LIN {X 0,Y 574.636,Z 652.296,A -85,B 0,C 180,E1 -2267.181,E2 -2267.181} C_VEL
LIN {X 0,Y 574.744,Z 636.733,A -85,B 0,C 180,E1 -2267.487,E2 -2267.487} C_VEL
LIN {X 0,Y 575.18,Z 481.073,A -85,B 0,C 180,E1 -2269.488,E2 -2269.488} C_VEL
LIN {X 0,Y 574.004,Z 474.783,A -85,B 0,C 180,E1 -2269.626,E2 -2269.626} C_VEL
LIN {X 0,Y 574.349,Z 449.397,A -85,B 0,C 180,E1 -2272.671,E2 -2272.671} C_VEL
LIN {X 0,Y 574.64,Z 427.548,A -85,B 0,C 180,E1 -2275.344,E2 -2275.344} C_VEL
LIN {X 0,Y 574.378,Z 424.427,A -85,B 0,C 180,E1 -2275.745,E2 -2275.745} C_VEL
LIN {X 0,Y 573.261,Z 419.708,A -85,B 0,C 180,E1 -2276.421,E2 -2276.421} C_VEL
LIN {X 0,Y 573.237,Z 419.708,A -85,B 0,C 180,E1 -2278.564,E2 -2278.564} C_VEL
LIN {X 0,Y 573.234,Z 419.702,A -85,B 0,C 180,E1 -2280.992,E2 -2280.992} C_VEL
LIN {X 0,Y 573.259,Z 419.698,A -85,B 0,C 180,E1 -2283.523,E2 -2283.523} C_VEL
LIN {X 0,Y 573.241,Z 419.705,A -85,B 0,C 180,E1 -2286.049,E2 -2286.049} C_VEL
LIN {X 0,Y 573.245,Z 419.702,A -85,B 0,C 180,E1 -2288.7,E2 -2288.7} C_VEL
LIN {X 0,Y 573.249,Z 419.699,A -85,B 0,C 180,E1 -2291.595,E2 -2291.595} C_VEL
LIN {X 0,Y 573.234,Z 419.71,A -85,B 0,C 180,E1 -2294.332,E2 -2294.332} C_VEL
LIN {X 0,Y 573.234,Z 419.699,A -85,B 0,C 180,E1 -2297.358,E2 -2297.358} C_VEL
LIN {X 0,Y 573.243,Z 419.708,A -85,B 0,C 180,E1 -2300.393,E2 -2300.393} C_VEL
LIN {X 0,Y 573.25,Z 419.698,A -85,B 0,C 180,E1 -2303.077,E2 -2303.077} C_VEL
LIN {X 0,Y 573.268,Z 419.697,A -85,B 0,C 180,E1 -2305.672,E2 -2305.672} C_VEL
LIN {X 0,Y 573.243,Z 419.706,A -85,B 0,C 180,E1 -2308.185,E2 -2308.185} C_VEL
LIN {X 0,Y 573.26,Z 419.702,A -85,B 0,C 180,E1 -2310.634,E2 -2310.634} C_VEL
LIN {X 0,Y 573.264,Z 419.696,A -85,B 0,C 180,E1 -2313.5,E2 -2313.5} C_VEL
LIN {X 0,Y 573.226,Z 419.707,A -85,B 0,C 180,E1 -2316.134,E2 -2316.134} C_VEL
LIN {X 0,Y 573.254,Z 419.697,A -85,B 0,C 180,E1 -2319.174,E2 -2319.174} C_VEL
LIN {X 0,Y 573.231,Z 419.7,A -85,B 0,C 180,E1 -2321.412,E2 -2321.412} C_VEL
LIN {X 0,Y 573.252,Z 419.697,A -85,B 0,C 180,E1 -2323.622,E2 -2323.622} C_VEL
LIN {X 0,Y 573.23,Z 419.707,A -85,B 0,C 180,E1 -2326.53,E2 -2326.53} C_VEL
LIN {X 0,Y 573.254,Z 419.701,A -85,B 0,C 180,E1 -2328.745,E2 -2328.745} C_VEL
LIN {X 0,Y 573.301,Z 419.691,A -85,B 0,C 180,E1 -2331.541,E2 -2331.541} C_VEL
LIN {X 0,Y 573.284,Z 419.703,A -85,B 0,C 180,E1 -2334.372,E2 -2334.372} C_VEL
LIN {X 0,Y 573.304,Z 419.693,A -85,B 0,C 180,E1 -2337.893,E2 -2337.893} C_VEL
LIN {X 0,Y 573.329,Z 419.692,A -85,B 0,C 180,E1 -2340.703,E2 -2340.703} C_VEL
LIN {X 0,Y 573.234,Z 419.7,A -85,B 0,C 180,E1 -2343.515,E2 -2343.515} C_VEL
LIN {X 0,Y 573.291,Z 419.693,A -85,B 0,C 180,E1 -2345.628,E2 -2345.628} C_VEL
LIN {X 0,Y 573.301,Z 419.701,A -85,B 0,C 180,E1 -2348.459,E2 -2348.459} C_VEL
LIN {X 0,Y 573.264,Z 419.695,A -85,B 0,C 180,E1 -2351.312,E2 -2351.312} C_VEL
LIN {X 0,Y 573.266,Z 419.702,A -85,B 0,C 180,E1 -2354.193,E2 -2354.193} C_VEL
LIN {X 0,Y 573.254,Z 419.698,A -85,B 0,C 180,E1 -2357.112,E2 -2357.112} C_VEL
LIN {X 0,Y 573.252,Z 419.702,A -85,B 0,C 180,E1 -2360.077,E2 -2360.077} C_VEL
LIN {X 0,Y 573.236,Z 419.709,A -85,B 0,C 180,E1 -2362.338,E2 -2362.338} C_VEL
LIN {X 0,Y 573.246,Z 419.703,A -85,B 0,C 180,E1 -2364.399,E2 -2364.399} C_VEL
LIN {X 0,Y 572.62,Z 419.784,A -85,B 0,C 180,E1 -2364.986,E2 -2364.986} C_VEL
LIN {X 0,Y 569.782,Z 420.136,A -85,B 0,C 180,E1 -2365.938,E2 -2365.938} C_VEL
LIN {X 0,Y 567.354,Z 420.438,A -85,B 0,C 180,E1 -2366.704,E2 -2366.704} C_VEL
LIN {X 0,Y 566.301,Z 420.564,A -85,B 0,C 180,E1 -2367.295,E2 -2367.295} C_VEL
LIN {X 0,Y 566.212,Z 420.575,A -85,B 0,C 180,E1 -2367.495,E2 -2367.495} C_VEL
LIN {X 0,Y 566.223,Z 420.574,A -85,B 0,C 180,E1 -2369.768,E2 -2369.768} C_VEL
LIN {X 0,Y 566.205,Z 420.584,A -85,B 0,C 180,E1 -2372.432,E2 -2372.432} C_VEL
LIN {X 0,Y 566.21,Z 420.578,A -85,B 0,C 180,E1 -2374.995,E2 -2374.995} C_VEL
LIN {X 0,Y 566.193,Z 420.578,A -85,B 0,C 180,E1 -2377.461,E2 -2377.461} C_VEL
LIN {X 0,Y 566.224,Z 420.581,A -85,B 0,C 180,E1 -2380.198,E2 -2380.198} C_VEL
LIN {X 0,Y 566.198,Z 420.582,A -85,B 0,C 180,E1 -2383.055,E2 -2383.055} C_VEL
LIN {X 0,Y 566.226,Z 420.717,A -85,B 0,C 180,E1 -2384.592,E2 -2384.592} C_VEL
LIN {X 0,Y 567.225,Z 426.295,A -85,B 0,C 180,E1 -2385.433,E2 -2385.433} C_VEL
LIN {X 0,Y 566.895,Z 445.97,A -85,B 0,C 180,E1 -2388.193,E2 -2388.193} C_VEL
LIN {X 0,Y 568.518,Z 454.109,A -85,B 0,C 180,E1 -2388.359,E2 -2388.359} C_VEL
LIN {X 0,Y 567.983,Z 611.267,A -85,B 0,C 180,E1 -2390.415,E2 -2390.415} C_VEL
LIN {X 0,Y 567.818,Z 627.039,A -85,B 0,C 180,E1 -2390.774,E2 -2390.774} C_VEL
LIN {X 0,Y 567.61,Z 641.985,A -85,B 0,C 180,E1 -2391.265,E2 -2391.265} C_VEL
LIN {X 0,Y 567.394,Z 656.381,A -85,B 0,C 180,E1 -2391.892,E2 -2391.892} C_VEL
LIN {X 0,Y 567.139,Z 669.582,A -85,B 0,C 180,E1 -2392.613,E2 -2392.613} C_VEL
LIN {X 0,Y 566.915,Z 682.658,A -85,B 0,C 180,E1 -2393.485,E2 -2393.485} C_VEL
LIN {X 0,Y 566.723,Z 693.514,A -85,B 0,C 180,E1 -2394.35,E2 -2394.35} C_VEL
LIN {X 0,Y 566.452,Z 704.885,A -85,B 0,C 180,E1 -2395.416,E2 -2395.416} C_VEL
LIN {X 0,Y 566.33,Z 714.474,A -85,B 0,C 180,E1 -2396.481,E2 -2396.481} C_VEL
LIN {X 0,Y 566.203,Z 724.073,A -85,B 0,C 180,E1 -2397.743,E2 -2397.743} C_VEL
LIN {X 0,Y 566.055,Z 731.777,A -85,B 0,C 180,E1 -2398.947,E2 -2398.947} C_VEL
LIN {X 0,Y 566.009,Z 739.23,A -85,B 0,C 180,E1 -2400.363,E2 -2400.363} C_VEL
LIN {X 0,Y 565.929,Z 745.455,A -85,B 0,C 180,E1 -2401.85,E2 -2401.85} C_VEL
LIN {X 0,Y 565.901,Z 750.37,A -85,B 0,C 180,E1 -2403.404,E2 -2403.404} C_VEL
LIN {X 0,Y 565.853,Z 753.908,A -85,B 0,C 180,E1 -2405.022,E2 -2405.022} C_VEL
LIN {X 0,Y 565.848,Z 755.883,A -85,B 0,C 180,E1 -2406.582,E2 -2406.582} C_VEL
LIN {X 0,Y 565.831,Z 756.489,A -85,B 0,C 180,E1 -2408.123,E2 -2408.123} C_VEL
LIN {X 0,Y 565.833,Z 755.776,A -85,B 0,C 180,E1 -2409.649,E2 -2409.649} C_VEL
LIN {X 0,Y 565.851,Z 753.765,A -85,B 0,C 180,E1 -2411.161,E2 -2411.161} C_VEL
LIN {X 0,Y 565.862,Z 750.442,A -85,B 0,C 180,E1 -2412.658,E2 -2412.658} C_VEL
LIN {X 0,Y 565.916,Z 745.782,A -85,B 0,C 180,E1 -2414.145,E2 -2414.145} C_VEL
LIN {X 0,Y 566.005,Z 739.706,A -85,B 0,C 180,E1 -2415.621,E2 -2415.621} C_VEL
LIN {X 0,Y 566.037,Z 732.099,A -85,B 0,C 180,E1 -2417.086,E2 -2417.086} C_VEL
LIN {X 0,Y 566.205,Z 723.96,A -85,B 0,C 180,E1 -2418.364,E2 -2418.364} C_VEL
LIN {X 0,Y 566.34,Z 714.266,A -85,B 0,C 180,E1 -2419.634,E2 -2419.634} C_VEL
LIN {X 0,Y 566.521,Z 704.419,A -85,B 0,C 180,E1 -2420.72,E2 -2420.72} C_VEL
LIN {X 0,Y 566.736,Z 692.793,A -85,B 0,C 180,E1 -2421.802,E2 -2421.802} C_VEL
LIN {X 0,Y 566.935,Z 680.459,A -85,B 0,C 180,E1 -2422.762,E2 -2422.762} C_VEL
LIN {X 0,Y 567.195,Z 667.503,A -85,B 0,C 180,E1 -2423.598,E2 -2423.598} C_VEL
LIN {X 0,Y 567.46,Z 653.878,A -85,B 0,C 180,E1 -2424.314,E2 -2424.314} C_VEL
LIN {X 0,Y 567.64,Z 640.029,A -85,B 0,C 180,E1 -2424.895,E2 -2424.895} C_VEL
LIN {X 0,Y 567.851,Z 625.202,A -85,B 0,C 180,E1 -2425.364,E2 -2425.364} C_VEL
LIN {X 0,Y 567.962,Z 609.905,A -85,B 0,C 180,E1 -2425.698,E2 -2425.698} C_VEL
LIN {X 0,Y 568.45,Z 453.464,A -85,B 0,C 180,E1 -2427.742,E2 -2427.742} C_VEL
LIN {X 0,Y 566.942,Z 445.815,A -85,B 0,C 180,E1 -2427.914,E2 -2427.914} C_VEL
LIN {X 0,Y 567.186,Z 425.932,A -85,B 0,C 180,E1 -2430.71,E2 -2430.71} C_VEL
LIN {X 0,Y 566.227,Z 420.583,A -85,B 0,C 180,E1 -2431.534,E2 -2431.534} C_VEL
LIN {X 0,Y 566.195,Z 420.587,A -85,B 0,C 180,E1 -2433.559,E2 -2433.559} C_VEL
LIN {X 0,Y 566.26,Z 420.577,A -85,B 0,C 180,E1 -2435.699,E2 -2435.699} C_VEL
LIN {X 0,Y 566.232,Z 420.573,A -85,B 0,C 180,E1 -2438.566,E2 -2438.566} C_VEL
LIN {X 0,Y 566.247,Z 420.575,A -85,B 0,C 180,E1 -2441.454,E2 -2441.454} C_VEL
LIN {X 0,Y 566.24,Z 420.572,A -85,B 0,C 180,E1 -2444.507,E2 -2444.507} C_VEL
LIN {X 0,Y 566.204,Z 420.581,A -85,B 0,C 180,E1 -2447.332,E2 -2447.332} C_VEL
LIN {X 0,Y 566.217,Z 420.575,A -85,B 0,C 180,E1 -2450.337,E2 -2450.337} C_VEL
LIN {X 0,Y 566.194,Z 420.583,A -85,B 0,C 180,E1 -2453.404,E2 -2453.404} C_VEL
LIN {X 0,Y 566.219,Z 420.582,A -85,B 0,C 180,E1 -2455.749,E2 -2455.749} C_VEL
LIN {X 0,Y 566.207,Z 420.576,A -85,B 0,C 180,E1 -2458.202,E2 -2458.202} C_VEL
LIN {X 0,Y 566.203,Z 420.578,A -85,B 0,C 180,E1 -2461.078,E2 -2461.078} C_VEL
LIN {X 0,Y 566.215,Z 420.583,A -85,B 0,C 180,E1 -2463.734,E2 -2463.734} C_VEL
LIN {X 0,Y 566.218,Z 420.573,A -85,B 0,C 180,E1 -2466.569,E2 -2466.569} C_VEL
LIN {X 0,Y 566.215,Z 420.584,A -85,B 0,C 180,E1 -2469.685,E2 -2469.685} C_VEL
LIN {X 0,Y 566.217,Z 420.576,A -85,B 0,C 180,E1 -2472.087,E2 -2472.087} C_VEL
LIN {X 0,Y 566.176,Z 420.58,A -85,B 0,C 180,E1 -2475.036,E2 -2475.036} C_VEL
LIN {X 0,Y 566.214,Z 420.575,A -85,B 0,C 180,E1 -2478.136,E2 -2478.136} C_VEL
LIN {X 0,Y 566.224,Z 420.573,A -85,B 0,C 180,E1 -2480.727,E2 -2480.727} C_VEL
LIN {X 0,Y 566.22,Z 420.58,A -85,B 0,C 180,E1 -2483.783,E2 -2483.783} C_VEL
LIN {X 0,Y 566.214,Z 420.576,A -85,B 0,C 180,E1 -2486.265,E2 -2486.265} C_VEL
LIN {X 0,Y 566.192,Z 420.577,A -85,B 0,C 180,E1 -2488.923,E2 -2488.923} C_VEL
LIN {X 0,Y 566.23,Z 420.579,A -85,B 0,C 180,E1 -2491.858,E2 -2491.858} C_VEL
LIN {X 0,Y 566.226,Z 420.574,A -85,B 0,C 180,E1 -2494.251,E2 -2494.251} C_VEL
LIN {X 0,Y 566.173,Z 420.576,A -85,B 0,C 180,E1 -2496.718,E2 -2496.718} C_VEL
LIN {X 0,Y 566.215,Z 420.584,A -85,B 0,C 180,E1 -2499.663,E2 -2499.663} C_VEL
LIN {X 0,Y 566.2,Z 420.574,A -85,B 0,C 180,E1 -2502.668,E2 -2502.668} C_VEL
LIN {X 0,Y 566.234,Z 420.58,A -85,B 0,C 180,E1 -2505.627,E2 -2505.627} C_VEL
LIN {X 0,Y 566.234,Z 420.57,A -85,B 0,C 180,E1 -2508.675,E2 -2508.675} C_VEL
LIN {X 0,Y 566.234,Z 420.575,A -85,B 0,C 180,E1 -2511.434,E2 -2511.434} C_VEL
LIN {X 0,Y 566.258,Z 420.57,A -85,B 0,C 180,E1 -2514.301,E2 -2514.301} C_VEL
LIN {X 0,Y 566.28,Z 420.572,A -85,B 0,C 180,E1 -2517.866,E2 -2517.866} C_VEL
LIN {X 0,Y 566.303,Z 420.563,A -85,B 0,C 180,E1 -2520.711,E2 -2520.711} C_VEL
LIN {X 0,Y 566.275,Z 420.566,A -85,B 0,C 180,E1 -2522.845,E2 -2522.845} C_VEL
LIN {X 0,Y 566.257,Z 420.576,A -85,B 0,C 180,E1 -2525.698,E2 -2525.698} C_VEL
LIN {X 0,Y 566.233,Z 420.572,A -85,B 0,C 180,E1 -2528.565,E2 -2528.565} C_VEL
LIN {X 0,Y 566.241,Z 420.575,A -85,B 0,C 180,E1 -2531.454,E2 -2531.454} C_VEL
LIN {X 0,Y 566.233,Z 420.572,A -85,B 0,C 180,E1 -2534.506,E2 -2534.506} C_VEL
LIN {X 0,Y 566.199,Z 420.58,A -85,B 0,C 180,E1 -2537.331,E2 -2537.331} C_VEL
LIN {X 0,Y 566.213,Z 420.576,A -85,B 0,C 180,E1 -2540.337,E2 -2540.337} C_VEL
LIN {X 0,Y 566.188,Z 420.582,A -85,B 0,C 180,E1 -2543.404,E2 -2543.404} C_VEL
LIN {X 0,Y 566.215,Z 420.584,A -85,B 0,C 180,E1 -2545.749,E2 -2545.749} C_VEL
LIN {X 0,Y 566.205,Z 420.578,A -85,B 0,C 180,E1 -2548.203,E2 -2548.203} C_VEL
LIN {X 0,Y 566.189,Z 420.578,A -85,B 0,C 180,E1 -2551.076,E2 -2551.076} C_VEL
LIN {X 0,Y 566.212,Z 420.584,A -85,B 0,C 180,E1 -2553.734,E2 -2553.734} C_VEL
LIN {X 0,Y 566.216,Z 420.574,A -85,B 0,C 180,E1 -2556.569,E2 -2556.569} C_VEL
LIN {X 0,Y 566.211,Z 420.585,A -85,B 0,C 180,E1 -2559.685,E2 -2559.685} C_VEL
LIN {X 0,Y 566.188,Z 420.582,A -85,B 0,C 180,E1 -2562.09,E2 -2562.09} C_VEL
LIN {X 0,Y 566.174,Z 420.58,A -85,B 0,C 180,E1 -2565.036,E2 -2565.036} C_VEL
LIN {X 0,Y 566.214,Z 420.582,A -85,B 0,C 180,E1 -2567.913,E2 -2567.913} C_VEL
LIN {X 0,Y 566.217,Z 420.574,A -85,B 0,C 180,E1 -2570.727,E2 -2570.727} C_VEL
LIN {X 0,Y 566.184,Z 420.587,A -85,B 0,C 180,E1 -2573.788,E2 -2573.788} C_VEL
LIN {X 0,Y 566.212,Z 420.579,A -85,B 0,C 180,E1 -2576.266,E2 -2576.266} C_VEL
LIN {X 0,Y 566.196,Z 420.579,A -85,B 0,C 180,E1 -2578.923,E2 -2578.923} C_VEL
LIN {X 0,Y 566.212,Z 420.585,A -85,B 0,C 180,E1 -2581.857,E2 -2581.857} C_VEL
LIN {X 0,Y 566.204,Z 420.669,A -85,B 0,C 180,E1 -2583.394,E2 -2583.394} C_VEL
LIN {X 0,Y 567.792,Z 427.532,A -85,B 0,C 180,E1 -2584.328,E2 -2584.328} C_VEL
LIN {X 0,Y 567.557,Z 447.83,A -85,B 0,C 180,E1 -2586.849,E2 -2586.849} C_VEL
LIN {X 0,Y 567.148,Z 472.644,A -85,B 0,C 180,E1 -2589.868,E2 -2589.868} C_VEL
LIN {X 0,Y 567.114,Z 474.917,A -85,B 0,C 180,E1 -2590.142,E2 -2590.142} C_VEL
LIN {X 0,Y 568.492,Z 482.253,A -85,B 0,C 180,E1 -2590.289,E2 -2590.289} C_VEL
LIN {X 0,Y 567.986,Z 640.908,A -85,B 0,C 180,E1 -2592.363,E2 -2592.363} C_VEL
LIN {X 0,Y 567.836,Z 656.698,A -85,B 0,C 180,E1 -2592.72,E2 -2592.72} C_VEL
LIN {X 0,Y 567.632,Z 672.035,A -85,B 0,C 180,E1 -2593.223,E2 -2593.223} C_VEL
LIN {X 0,Y 567.459,Z 685.767,A -85,B 0,C 180,E1 -2593.819,E2 -2593.819} C_VEL
LIN {X 0,Y 567.151,Z 699.241,A -85,B 0,C 180,E1 -2594.548,E2 -2594.548} C_VEL
LIN {X 0,Y 566.932,Z 711.516,A -85,B 0,C 180,E1 -2595.359,E2 -2595.359} C_VEL
LIN {X 0,Y 566.672,Z 724.287,A -85,B 0,C 180,E1 -2596.37,E2 -2596.37} C_VEL
LIN {X 0,Y 566.491,Z 735.746,A -85,B 0,C 180,E1 -2597.461,E2 -2597.461} C_VEL
LIN {X 0,Y 566.269,Z 746.31,A -85,B 0,C 180,E1 -2598.659,E2 -2598.659} C_VEL
LIN {X 0,Y 566.208,Z 754.855,A -85,B 0,C 180,E1 -2599.812,E2 -2599.812} C_VEL
LIN {X 0,Y 566.058,Z 762.732,A -85,B 0,C 180,E1 -2601.072,E2 -2601.072} C_VEL
LIN {X 0,Y 565.998,Z 770.088,A -85,B 0,C 180,E1 -2602.508,E2 -2602.508} C_VEL
LIN {X 0,Y 565.956,Z 775.922,A -85,B 0,C 180,E1 -2603.941,E2 -2603.941} C_VEL
LIN {X 0,Y 565.866,Z 779.384,A -85,B 0,C 180,E1 -2605.012,E2 -2605.012} C_VEL
LIN {X 0,Y 565.909,Z 782.889,A -85,B 0,C 180,E1 -2606.44,E2 -2606.44} C_VEL
LIN {X 0,Y 565.836,Z 785.192,A -85,B 0,C 180,E1 -2607.864,E2 -2607.864} C_VEL
LIN {X 0,Y 565.838,Z 786.349,A -85,B 0,C 180,E1 -2609.288,E2 -2609.288} C_VEL
LIN {X 0,Y 565.838,Z 786.349,A -85,B 0,C 180,E1 -2610.711,E2 -2610.711} C_VEL
LIN {X 0,Y 565.836,Z 785.191,A -85,B 0,C 180,E1 -2612.135,E2 -2612.135} C_VEL
LIN {X 0,Y 565.909,Z 782.888,A -85,B 0,C 180,E1 -2613.56,E2 -2613.56} C_VEL
LIN {X 0,Y 565.866,Z 779.387,A -85,B 0,C 180,E1 -2614.987,E2 -2614.987} C_VEL
LIN {X 0,Y 565.956,Z 775.926,A -85,B 0,C 180,E1 -2616.059,E2 -2616.059} C_VEL
LIN {X 0,Y 565.999,Z 770.09,A -85,B 0,C 180,E1 -2617.491,E2 -2617.491} C_VEL
LIN {X 0,Y 566.057,Z 762.733,A -85,B 0,C 180,E1 -2618.928,E2 -2618.928} C_VEL
LIN {X 0,Y 566.208,Z 754.86,A -85,B 0,C 180,E1 -2620.187,E2 -2620.187} C_VEL
LIN {X 0,Y 566.307,Z 745.395,A -85,B 0,C 180,E1 -2621.452,E2 -2621.452} C_VEL
LIN {X 0,Y 566.491,Z 735.754,A -85,B 0,C 180,E1 -2622.539,E2 -2622.539} C_VEL
LIN {X 0,Y 566.671,Z 724.3,A -85,B 0,C 180,E1 -2623.629,E2 -2623.629} C_VEL
LIN {X 0,Y 566.926,Z 711.683,A -85,B 0,C 180,E1 -2624.63,E2 -2624.63} C_VEL
LIN {X 0,Y 567.123,Z 699.253,A -85,B 0,C 180,E1 -2625.452,E2 -2625.452} C_VEL
LIN {X 0,Y 567.418,Z 685.779,A -85,B 0,C 180,E1 -2626.181,E2 -2626.181} C_VEL
LIN {X 0,Y 567.606,Z 672.062,A -85,B 0,C 180,E1 -2626.777,E2 -2626.777} C_VEL
LIN {X 0,Y 567.845,Z 656.738,A -85,B 0,C 180,E1 -2627.279,E2 -2627.279} C_VEL
LIN {X 0,Y 567.978,Z 641.331,A -85,B 0,C 180,E1 -2627.629,E2 -2627.629} C_VEL
LIN {X 0,Y 568.463,Z 481.789,A -85,B 0,C 180,E1 -2629.718,E2 -2629.718} C_VEL
LIN {X 0,Y 567.132,Z 474.839,A -85,B 0,C 180,E1 -2629.867,E2 -2629.867} C_VEL
LIN {X 0,Y 567.488,Z 449.397,A -85,B 0,C 180,E1 -2632.961,E2 -2632.961} C_VEL
LIN {X 0,Y 567.849,Z 429.252,A -85,B 0,C 180,E1 -2635.454,E2 -2635.454} C_VEL
LIN {X 0,Y 567.492,Z 425.948,A -85,B 0,C 180,E1 -2635.883,E2 -2635.883} C_VEL
LIN {X 0,Y 566.205,Z 420.587,A -85,B 0,C 180,E1 -2636.626,E2 -2636.626} C_VEL
LIN {X 0,Y 566.19,Z 420.582,A -85,B 0,C 180,E1 -2638.953,E2 -2638.953} C_VEL
LIN {X 0,Y 566.199,Z 420.578,A -85,B 0,C 180,E1 -2641.421,E2 -2641.421} C_VEL
LIN {X 0,Y 566.206,Z 420.581,A -85,B 0,C 180,E1 -2643.955,E2 -2643.955} C_VEL
LIN {X 0,Y 566.208,Z 420.581,A -85,B 0,C 180,E1 -2646.568,E2 -2646.568} C_VEL
LIN {X 0,Y 566.209,Z 420.577,A -85,B 0,C 180,E1 -2649.685,E2 -2649.685} C_VEL
LIN {X 0,Y 566.212,Z 420.582,A -85,B 0,C 180,E1 -2652.086,E2 -2652.086} C_VEL
LIN {X 0,Y 566.168,Z 420.581,A -85,B 0,C 180,E1 -2655.035,E2 -2655.035} C_VEL
LIN {X 0,Y 566.212,Z 420.581,A -85,B 0,C 180,E1 -2658.135,E2 -2658.135} C_VEL
LIN {X 0,Y 566.217,Z 420.578,A -85,B 0,C 180,E1 -2660.727,E2 -2660.727} C_VEL
LIN {X 0,Y 566.212,Z 420.577,A -85,B 0,C 180,E1 -2663.783,E2 -2663.783} C_VEL
LIN {X 0,Y 566.223,Z 420.583,A -85,B 0,C 180,E1 -2666.263,E2 -2666.263} C_VEL
LIN {X 0,Y 566.192,Z 420.578,A -85,B 0,C 180,E1 -2668.922,E2 -2668.922} C_VEL
LIN {X 0,Y 566.221,Z 420.576,A -85,B 0,C 180,E1 -2671.858,E2 -2671.858} C_VEL
LIN {X 0,Y 566.22,Z 420.582,A -85,B 0,C 180,E1 -2674.251,E2 -2674.251} C_VEL
LIN {X 0,Y 566.184,Z 420.582,A -85,B 0,C 180,E1 -2676.713,E2 -2676.713} C_VEL
LIN {X 0,Y 566.212,Z 420.575,A -85,B 0,C 180,E1 -2679.663,E2 -2679.663} C_VEL
LIN {X 0,Y 566.197,Z 420.58,A -85,B 0,C 180,E1 -2682.668,E2 -2682.668} C_VEL
LIN {X 0,Y 566.226,Z 420.573,A -85,B 0,C 180,E1 -2685.627,E2 -2685.627} C_VEL
LIN {X 0,Y 566.226,Z 420.577,A -85,B 0,C 180,E1 -2688.675,E2 -2688.675} C_VEL
LIN {X 0,Y 566.242,Z 420.57,A -85,B 0,C 180,E1 -2691.435,E2 -2691.435} C_VEL
LIN {X 0,Y 566.252,Z 420.578,A -85,B 0,C 180,E1 -2694.302,E2 -2694.302} C_VEL
LIN {X 0,Y 566.275,Z 420.568,A -85,B 0,C 180,E1 -2697.866,E2 -2697.866} C_VEL
LIN {X 0,Y 566.299,Z 420.567,A -85,B 0,C 180,E1 -2700.711,E2 -2700.711} C_VEL
LIN {X 0,Y 566.272,Z 420.57,A -85,B 0,C 180,E1 -2702.846,E2 -2702.846} C_VEL
LIN {X 0,Y 566.26,Z 420.569,A -85,B 0,C 180,E1 -2705.698,E2 -2705.698} C_VEL
LIN {X 0,Y 566.242,Z 420.578,A -85,B 0,C 180,E1 -2708.566,E2 -2708.566} C_VEL
LIN {X 0,Y 566.234,Z 420.571,A -85,B 0,C 180,E1 -2711.455,E2 -2711.455} C_VEL
LIN {X 0,Y 566.227,Z 420.581,A -85,B 0,C 180,E1 -2714.507,E2 -2714.507} C_VEL
LIN {X 0,Y 566.199,Z 420.576,A -85,B 0,C 180,E1 -2717.332,E2 -2717.332} C_VEL
LIN {X 0,Y 566.214,Z 420.583,A -85,B 0,C 180,E1 -2720.337,E2 -2720.337} C_VEL
LIN {X 0,Y 566.185,Z 420.578,A -85,B 0,C 180,E1 -2723.404,E2 -2723.404} C_VEL
LIN {X 0,Y 566.222,Z 420.575,A -85,B 0,C 180,E1 -2725.749,E2 -2725.749} C_VEL
LIN {X 0,Y 566.212,Z 420.575,A -85,B 0,C 180,E1 -2727.495,E2 -2727.495} C_VEL
LIN {X 0,Y 565.534,Z 420.666,A -85,B 0,C 180,E1 -2728.089,E2 -2728.089} C_VEL
LIN {X 0,Y 562.669,Z 421.02,A -85,B 0,C 180,E1 -2729.053,E2 -2729.053} C_VEL
LIN {X 0,Y 560.258,Z 421.32,A -85,B 0,C 180,E1 -2729.828,E2 -2729.828} C_VEL
LIN {X 0,Y 559.229,Z 421.453,A -85,B 0,C 180,E1 -2730.427,E2 -2730.427} C_VEL
LIN {X 0,Y 559.148,Z 421.457,A -85,B 0,C 180,E1 -2730.63,E2 -2730.63} C_VEL
LIN {X 0,Y 559.174,Z 421.452,A -85,B 0,C 180,E1 -2733.574,E2 -2733.574} C_VEL
LIN {X 0,Y 559.186,Z 421.459,A -85,B 0,C 180,E1 -2736.452,E2 -2736.452} C_VEL
LIN {X 0,Y 559.175,Z 421.456,A -85,B 0,C 180,E1 -2738.934,E2 -2738.934} C_VEL
LIN {X 0,Y 559.188,Z 421.452,A -85,B 0,C 180,E1 -2741.768,E2 -2741.768} C_VEL
LIN {X 0,Y 559.173,Z 421.48,A -85,B 0,C 180,E1 -2744.381,E2 -2744.381} C_VEL
LIN {X 0,Y 560.333,Z 427.983,A -85,B 0,C 180,E1 -2745.383,E2 -2745.383} C_VEL
LIN {X 0,Y 560.011,Z 446.073,A -85,B 0,C 180,E1 -2747.94,E2 -2747.94} C_VEL
LIN {X 0,Y 561.851,Z 454.621,A -85,B 0,C 180,E1 -2748.122,E2 -2748.122} C_VEL
LIN {X 0,Y 561.246,Z 610.539,A -85,B 0,C 180,E1 -2750.183,E2 -2750.183} C_VEL
LIN {X 0,Y 561.067,Z 625.756,A -85,B 0,C 180,E1 -2750.524,E2 -2750.524} C_VEL
LIN {X 0,Y 560.791,Z 641.157,A -85,B 0,C 180,E1 -2751.024,E2 -2751.024} C_VEL
LIN {X 0,Y 560.602,Z 655.412,A -85,B 0,C 180,E1 -2751.644,E2 -2751.644} C_VEL
LIN {X 0,Y 560.268,Z 669.518,A -85,B 0,C 180,E1 -2752.415,E2 -2752.415} C_VEL
LIN {X 0,Y 560.003,Z 681.869,A -85,B 0,C 180,E1 -2753.243,E2 -2753.243} C_VEL
LIN {X 0,Y 559.772,Z 693.455,A -85,B 0,C 180,E1 -2754.171,E2 -2754.171} C_VEL
LIN {X 0,Y 559.498,Z 704.848,A -85,B 0,C 180,E1 -2755.253,E2 -2755.253} C_VEL
LIN {X 0,Y 559.29,Z 715.295,A -85,B 0,C 180,E1 -2756.435,E2 -2756.435} C_VEL
LIN {X 0,Y 559.137,Z 724.751,A -85,B 0,C 180,E1 -2757.711,E2 -2757.711} C_VEL
LIN {X 0,Y 558.996,Z 732.557,A -85,B 0,C 180,E1 -2758.972,E2 -2758.972} C_VEL
LIN {X 0,Y 558.921,Z 739.865,A -85,B 0,C 180,E1 -2760.408,E2 -2760.408} C_VEL
LIN {X 0,Y 558.852,Z 745.129,A -85,B 0,C 180,E1 -2761.68,E2 -2761.68} C_VEL
LIN {X 0,Y 558.819,Z 750.115,A -85,B 0,C 180,E1 -2763.245,E2 -2763.245} C_VEL
LIN {X 0,Y 558.764,Z 753.784,A -85,B 0,C 180,E1 -2764.905,E2 -2764.905} C_VEL
LIN {X 0,Y 558.759,Z 755.949,A -85,B 0,C 180,E1 -2766.663,E2 -2766.663} C_VEL
LIN {X 0,Y 558.724,Z 756.46,A -85,B 0,C 180,E1 -2767.83,E2 -2767.83} C_VEL
LIN {X 0,Y 558.743,Z 755.982,A -85,B 0,C 180,E1 -2769.379,E2 -2769.379} C_VEL
LIN {X 0,Y 558.778,Z 754.211,A -85,B 0,C 180,E1 -2770.913,E2 -2770.913} C_VEL
LIN {X 0,Y 558.765,Z 751.149,A -85,B 0,C 180,E1 -2772.431,E2 -2772.431} C_VEL
LIN {X 0,Y 558.823,Z 746.756,A -85,B 0,C 180,E1 -2773.938,E2 -2773.938} C_VEL
LIN {X 0,Y 558.917,Z 740.963,A -85,B 0,C 180,E1 -2775.435,E2 -2775.435} C_VEL
LIN {X 0,Y 558.981,Z 733.656,A -85,B 0,C 180,E1 -2776.921,E2 -2776.921} C_VEL
LIN {X 0,Y 559.137,Z 725.854,A -85,B 0,C 180,E1 -2778.215,E2 -2778.215} C_VEL
LIN {X 0,Y 559.3,Z 716.529,A -85,B 0,C 180,E1 -2779.502,E2 -2779.502} C_VEL
LIN {X 0,Y 559.461,Z 707.123,A -85,B 0,C 180,E1 -2780.602,E2 -2780.602} C_VEL
LIN {X 0,Y 559.712,Z 695.993,A -85,B 0,C 180,E1 -2781.698,E2 -2781.698} C_VEL
LIN {X 0,Y 559.957,Z 683.762,A -85,B 0,C 180,E1 -2782.709,E2 -2782.709} C_VEL
LIN {X 0,Y 560.27,Z 670.608,A -85,B 0,C 180,E1 -2783.609,E2 -2783.609} C_VEL
LIN {X 0,Y 560.567,Z 655.887,A -85,B 0,C 180,E1 -2784.425,E2 -2784.425} C_VEL
LIN {X 0,Y 560.827,Z 641.346,A -85,B 0,C 180,E1 -2785.058,E2 -2785.058} C_VEL
LIN {X 0,Y 561.07,Z 626.158,A -85,B 0,C 180,E1 -2785.555,E2 -2785.555} C_VEL
LIN {X 0,Y 561.224,Z 611.314,A -85,B 0,C 180,E1 -2785.894,E2 -2785.894} C_VEL
LIN {X 0,Y 561.79,Z 454.392,A -85,B 0,C 180,E1 -2787.973,E2 -2787.973} C_VEL
LIN {X 0,Y 560.006,Z 445.905,A -85,B 0,C 180,E1 -2788.158,E2 -2788.158} C_VEL
LIN {X 0,Y 560.296,Z 427.911,A -85,B 0,C 180,E1 -2790.719,E2 -2790.719} C_VEL
LIN {X 0,Y 559.211,Z 421.457,A -85,B 0,C 180,E1 -2791.711,E2 -2791.711} C_VEL
LIN {X 0,Y 559.148,Z 421.464,A -85,B 0,C 180,E1 -2793.604,E2 -2793.604} C_VEL
LIN {X 0,Y 559.227,Z 421.453,A -85,B 0,C 180,E1 -2795.771,E2 -2795.771} C_VEL
LIN {X 0,Y 559.191,Z 421.451,A -85,B 0,C 180,E1 -2798.675,E2 -2798.675} C_VEL
LIN {X 0,Y 559.211,Z 421.454,A -85,B 0,C 180,E1 -2801.601,E2 -2801.601} C_VEL
LIN {X 0,Y 559.205,Z 421.448,A -85,B 0,C 180,E1 -2804.596,E2 -2804.596} C_VEL
LIN {X 0,Y 559.163,Z 421.462,A -85,B 0,C 180,E1 -2807.557,E2 -2807.557} C_VEL
LIN {X 0,Y 559.174,Z 421.458,A -85,B 0,C 180,E1 -2809.837,E2 -2809.837} C_VEL
LIN {X 0,Y 559.146,Z 421.458,A -85,B 0,C 180,E1 -2812.153,E2 -2812.153} C_VEL
LIN {X 0,Y 559.184,Z 421.452,A -85,B 0,C 180,E1 -2815.187,E2 -2815.187} C_VEL
LIN {X 0,Y 559.185,Z 421.457,A -85,B 0,C 180,E1 -2817.712,E2 -2817.712} C_VEL
LIN {X 0,Y 559.161,Z 421.455,A -85,B 0,C 180,E1 -2820.182,E2 -2820.182} C_VEL
LIN {X 0,Y 559.179,Z 421.448,A -85,B 0,C 180,E1 -2822.714,E2 -2822.714} C_VEL
LIN {X 0,Y 559.151,Z 421.459,A -85,B 0,C 180,E1 -2825.322,E2 -2825.322} C_VEL
LIN {X 0,Y 559.138,Z 421.458,A -85,B 0,C 180,E1 -2828.017,E2 -2828.017} C_VEL
LIN {X 0,Y 559.18,Z 421.451,A -85,B 0,C 180,E1 -2830.81,E2 -2830.81} C_VEL
LIN {X 0,Y 559.165,Z 421.461,A -85,B 0,C 180,E1 -2833.731,E2 -2833.731} C_VEL
LIN {X 0,Y 559.148,Z 421.454,A -85,B 0,C 180,E1 -2836.803,E2 -2836.803} C_VEL
LIN {X 0,Y 559.177,Z 421.452,A -85,B 0,C 180,E1 -2839.189,E2 -2839.189} C_VEL
LIN {X 0,Y 559.137,Z 421.46,A -85,B 0,C 180,E1 -2841.982,E2 -2841.982} C_VEL
LIN {X 0,Y 559.159,Z 421.451,A -85,B 0,C 180,E1 -2844.678,E2 -2844.678} C_VEL
LIN {X 0,Y 559.175,Z 421.456,A -85,B 0,C 180,E1 -2847.361,E2 -2847.361} C_VEL
LIN {X 0,Y 559.15,Z 421.455,A -85,B 0,C 180,E1 -2850.142,E2 -2850.142} C_VEL
LIN {X 0,Y 559.181,Z 421.452,A -85,B 0,C 180,E1 -2853.098,E2 -2853.098} C_VEL
LIN {X 0,Y 559.158,Z 421.46,A -85,B 0,C 180,E1 -2855.495,E2 -2855.495} C_VEL
LIN {X 0,Y 559.172,Z 421.451,A -85,B 0,C 180,E1 -2858.624,E2 -2858.624} C_VEL
LIN {X 0,Y 559.169,Z 421.452,A -85,B 0,C 180,E1 -2860.926,E2 -2860.926} C_VEL
LIN {X 0,Y 559.17,Z 421.456,A -85,B 0,C 180,E1 -2863.948,E2 -2863.948} C_VEL
LIN {X 0,Y 559.172,Z 421.454,A -85,B 0,C 180,E1 -2866.184,E2 -2866.184} C_VEL
LIN {X 0,Y 559.195,Z 421.449,A -85,B 0,C 180,E1 -2869.133,E2 -2869.133} C_VEL
LIN {X 0,Y 559.206,Z 421.451,A -85,B 0,C 180,E1 -2872.053,E2 -2872.053} C_VEL
LIN {X 0,Y 559.255,Z 421.441,A -85,B 0,C 180,E1 -2874.953,E2 -2874.953} C_VEL
LIN {X 0,Y 559.251,Z 421.448,A -85,B 0,C 180,E1 -2877.839,E2 -2877.839} C_VEL
LIN {X 0,Y 559.273,Z 421.439,A -85,B 0,C 180,E1 -2880.72,E2 -2880.72} C_VEL
LIN {X 0,Y 559.241,Z 421.442,A -85,B 0,C 180,E1 -2882.881,E2 -2882.881} C_VEL
LIN {X 0,Y 559.227,Z 421.452,A -85,B 0,C 180,E1 -2885.77,E2 -2885.77} C_VEL
LIN {X 0,Y 559.191,Z 421.449,A -85,B 0,C 180,E1 -2888.674,E2 -2888.674} C_VEL
LIN {X 0,Y 559.205,Z 421.454,A -85,B 0,C 180,E1 -2891.6,E2 -2891.6} C_VEL
LIN {X 0,Y 559.199,Z 421.448,A -85,B 0,C 180,E1 -2894.595,E2 -2894.595} C_VEL
LIN {X 0,Y 559.159,Z 421.46,A -85,B 0,C 180,E1 -2897.557,E2 -2897.557} C_VEL
LIN {X 0,Y 559.172,Z 421.459,A -85,B 0,C 180,E1 -2899.837,E2 -2899.837} C_VEL
LIN {X 0,Y 559.141,Z 421.458,A -85,B 0,C 180,E1 -2902.153,E2 -2902.153} C_VEL
LIN {X 0,Y 559.178,Z 421.453,A -85,B 0,C 180,E1 -2905.187,E2 -2905.187} C_VEL
LIN {X 0,Y 559.191,Z 421.459,A -85,B 0,C 180,E1 -2907.711,E2 -2907.711} C_VEL
LIN {X 0,Y 559.152,Z 421.456,A -85,B 0,C 180,E1 -2910.183,E2 -2910.183} C_VEL
LIN {X 0,Y 559.174,Z 421.451,A -85,B 0,C 180,E1 -2912.714,E2 -2912.714} C_VEL
LIN {X 0,Y 559.157,Z 421.457,A -85,B 0,C 180,E1 -2915.322,E2 -2915.322} C_VEL
LIN {X 0,Y 559.134,Z 421.461,A -85,B 0,C 180,E1 -2918.017,E2 -2918.017} C_VEL
LIN {X 0,Y 559.173,Z 421.451,A -85,B 0,C 180,E1 -2920.811,E2 -2920.811} C_VEL
LIN {X 0,Y 559.159,Z 421.463,A -85,B 0,C 180,E1 -2923.732,E2 -2923.732} C_VEL
LIN {X 0,Y 559.168,Z 421.452,A -85,B 0,C 180,E1 -2926.801,E2 -2926.801} C_VEL
LIN {X 0,Y 559.159,Z 421.456,A -85,B 0,C 180,E1 -2929.188,E2 -2929.188} C_VEL
LIN {X 0,Y 559.135,Z 421.462,A -85,B 0,C 180,E1 -2931.983,E2 -2931.983} C_VEL
LIN {X 0,Y 559.132,Z 421.458,A -85,B 0,C 180,E1 -2934.787,E2 -2934.787} C_VEL
LIN {X 0,Y 559.158,Z 421.46,A -85,B 0,C 180,E1 -2937.364,E2 -2937.364} C_VEL
LIN {X 0,Y 559.15,Z 421.462,A -85,B 0,C 180,E1 -2940.142,E2 -2940.142} C_VEL
LIN {X 0,Y 559.17,Z 421.459,A -85,B 0,C 180,E1 -2943.098,E2 -2943.098} C_VEL
LIN {X 0,Y 559.187,Z 421.563,A -85,B 0,C 180,E1 -2943.169,E2 -2943.169} C_VEL
LIN {X 0,Y 560.998,Z 429.565,A -85,B 0,C 180,E1 -2944.271,E2 -2944.271} C_VEL
LIN {X 0,Y 560.697,Z 449.39,A -85,B 0,C 180,E1 -2946.744,E2 -2946.744} C_VEL
LIN {X 0,Y 560.258,Z 473.295,A -85,B 0,C 180,E1 -2949.689,E2 -2949.689} C_VEL
LIN {X 0,Y 560.265,Z 475.041,A -85,B 0,C 180,E1 -2949.891,E2 -2949.891} C_VEL
LIN {X 0,Y 561.814,Z 483.76,A -85,B 0,C 180,E1 -2950.065,E2 -2950.065} C_VEL
LIN {X 0,Y 561.233,Z 640.998,A -85,B 0,C 180,E1 -2952.146,E2 -2952.146} C_VEL
LIN {X 0,Y 561.075,Z 656.22,A -85,B 0,C 180,E1 -2952.492,E2 -2952.492} C_VEL
LIN {X 0,Y 560.848,Z 670.791,A -85,B 0,C 180,E1 -2952.967,E2 -2952.967} C_VEL
LIN {X 0,Y 560.638,Z 683.8,A -85,B 0,C 180,E1 -2953.523,E2 -2953.523} C_VEL
LIN {X 0,Y 560.317,Z 697.675,A -85,B 0,C 180,E1 -2954.262,E2 -2954.262} C_VEL
LIN {X 0,Y 560.021,Z 711.517,A -85,B 0,C 180,E1 -2955.174,E2 -2955.174} C_VEL
LIN {X 0,Y 559.722,Z 724.289,A -85,B 0,C 180,E1 -2956.198,E2 -2956.198} C_VEL
LIN {X 0,Y 559.516,Z 735.747,A -85,B 0,C 180,E1 -2957.302,E2 -2957.302} C_VEL
LIN {X 0,Y 559.304,Z 745.388,A -85,B 0,C 180,E1 -2958.401,E2 -2958.401} C_VEL
LIN {X 0,Y 559.168,Z 754.854,A -85,B 0,C 180,E1 -2959.682,E2 -2959.682} C_VEL
LIN {X 0,Y 559.003,Z 762.733,A -85,B 0,C 180,E1 -2960.958,E2 -2960.958} C_VEL
LIN {X 0,Y 558.921,Z 770.088,A -85,B 0,C 180,E1 -2962.413,E2 -2962.413} C_VEL
LIN {X 0,Y 558.838,Z 775.306,A -85,B 0,C 180,E1 -2963.684,E2 -2963.684} C_VEL
LIN {X 0,Y 558.787,Z 779.385,A -85,B 0,C 180,E1 -2964.949,E2 -2964.949} C_VEL
LIN {X 0,Y 558.819,Z 782.889,A -85,B 0,C 180,E1 -2966.394,E2 -2966.394} C_VEL
LIN {X 0,Y 558.742,Z 785.191,A -85,B 0,C 180,E1 -2967.837,E2 -2967.837} C_VEL
LIN {X 0,Y 558.739,Z 786.349,A -85,B 0,C 180,E1 -2969.279,E2 -2969.279} C_VEL
LIN {X 0,Y 558.739,Z 786.348,A -85,B 0,C 180,E1 -2970.72,E2 -2970.72} C_VEL
LIN {X 0,Y 558.742,Z 785.19,A -85,B 0,C 180,E1 -2972.162,E2 -2972.162} C_VEL
LIN {X 0,Y 558.818,Z 782.887,A -85,B 0,C 180,E1 -2973.605,E2 -2973.605} C_VEL
LIN {X 0,Y 558.787,Z 779.387,A -85,B 0,C 180,E1 -2975.05,E2 -2975.05} C_VEL
LIN {X 0,Y 558.842,Z 774.61,A -85,B 0,C 180,E1 -2976.498,E2 -2976.498} C_VEL
LIN {X 0,Y 558.951,Z 768.425,A -85,B 0,C 180,E1 -2977.95,E2 -2977.95} C_VEL
LIN {X 0,Y 559.005,Z 760.65,A -85,B 0,C 180,E1 -2979.406,E2 -2979.406} C_VEL
LIN {X 0,Y 559.216,Z 752.372,A -85,B 0,C 180,E1 -2980.682,E2 -2980.682} C_VEL
LIN {X 0,Y 559.361,Z 742.396,A -85,B 0,C 180,E1 -2981.964,E2 -2981.964} C_VEL
LIN {X 0,Y 559.595,Z 732.193,A -85,B 0,C 180,E1 -2983.065,E2 -2983.065} C_VEL
LIN {X 0,Y 559.861,Z 720.026,A -85,B 0,C 180,E1 -2984.169,E2 -2984.169} C_VEL
LIN {X 0,Y 560.122,Z 707.698,A -85,B 0,C 180,E1 -2985.099,E2 -2985.099} C_VEL
LIN {X 0,Y 560.357,Z 694.522,A -85,B 0,C 180,E1 -2985.923,E2 -2985.923} C_VEL
LIN {X 0,Y 560.665,Z 679.841,A -85,B 0,C 180,E1 -2986.662,E2 -2986.662} C_VEL
LIN {X 0,Y 560.92,Z 665.632,A -85,B 0,C 180,E1 -2987.217,E2 -2987.217} C_VEL
LIN {X 0,Y 561.141,Z 651.171,A -85,B 0,C 180,E1 -2987.637,E2 -2987.637} C_VEL
LIN {X 0,Y 561.232,Z 636.68,A -85,B 0,C 180,E1 -2987.923,E2 -2987.923} C_VEL
LIN {X 0,Y 561.782,Z 482.838,A -85,B 0,C 180,E1 -2989.949,E2 -2989.949} C_VEL
LIN {X 0,Y 560.236,Z 474.914,A -85,B 0,C 180,E1 -2990.113,E2 -2990.113} C_VEL
LIN {X 0,Y 560.643,Z 450.958,A -85,B 0,C 180,E1 -2993.062,E2 -2993.062} C_VEL
LIN {X 0,Y 560.995,Z 429.549,A -85,B 0,C 180,E1 -2995.728,E2 -2995.728} C_VEL
LIN {X 0,Y 559.179,Z 421.46,A -85,B 0,C 180,E1 -2996.864,E2 -2996.864} C_VEL
LIN {X 0,Y 559.168,Z 421.46,A -85,B 0,C 180,E1 -2999.861,E2 -2999.861} C_VEL
LIN {X 0,Y 559.173,Z 421.456,A -85,B 0,C 180,E1 -3002.713,E2 -3002.713} C_VEL
LIN {X 0,Y 559.141,Z 421.456,A -85,B 0,C 180,E1 -3005.322,E2 -3005.322} C_VEL
LIN {X 0,Y 559.132,Z 421.462,A -85,B 0,C 180,E1 -3008.017,E2 -3008.017} C_VEL
LIN {X 0,Y 559.172,Z 421.455,A -85,B 0,C 180,E1 -3010.81,E2 -3010.81} C_VEL
LIN {X 0,Y 559.159,Z 421.454,A -85,B 0,C 180,E1 -3013.731,E2 -3013.731} C_VEL
LIN {X 0,Y 559.14,Z 421.457,A -85,B 0,C 180,E1 -3016.803,E2 -3016.803} C_VEL
LIN {X 0,Y 559.171,Z 421.452,A -85,B 0,C 180,E1 -3019.189,E2 -3019.189} C_VEL
LIN {X 0,Y 559.129,Z 421.462,A -85,B 0,C 180,E1 -3021.982,E2 -3021.982} C_VEL
LIN {X 0,Y 559.154,Z 421.457,A -85,B 0,C 180,E1 -3024.782,E2 -3024.782} C_VEL
LIN {X 0,Y 559.168,Z 421.451,A -85,B 0,C 180,E1 -3027.361,E2 -3027.361} C_VEL
LIN {X 0,Y 559.143,Z 421.462,A -85,B 0,C 180,E1 -3030.142,E2 -3030.142} C_VEL
LIN {X 0,Y 559.175,Z 421.451,A -85,B 0,C 180,E1 -3033.17,E2 -3033.17} C_VEL
LIN {X 0,Y 559.15,Z 421.454,A -85,B 0,C 180,E1 -3035.495,E2 -3035.495} C_VEL
LIN {X 0,Y 559.17,Z 421.456,A -85,B 0,C 180,E1 -3038.624,E2 -3038.624} C_VEL
LIN {X 0,Y 559.165,Z 421.454,A -85,B 0,C 180,E1 -3040.926,E2 -3040.926} C_VEL
LIN {X 0,Y 559.164,Z 421.455,A -85,B 0,C 180,E1 -3043.948,E2 -3043.948} C_VEL
LIN {X 0,Y 559.166,Z 421.459,A -85,B 0,C 180,E1 -3046.184,E2 -3046.184} C_VEL
LIN {X 0,Y 559.189,Z 421.45,A -85,B 0,C 180,E1 -3049.134,E2 -3049.134} C_VEL
LIN {X 0,Y 559.202,Z 421.452,A -85,B 0,C 180,E1 -3052.054,E2 -3052.054} C_VEL
LIN {X 0,Y 559.251,Z 421.443,A -85,B 0,C 180,E1 -3054.953,E2 -3054.953} C_VEL
LIN {X 0,Y 559.247,Z 421.444,A -85,B 0,C 180,E1 -3057.84,E2 -3057.84} C_VEL
LIN {X 0,Y 559.269,Z 421.443,A -85,B 0,C 180,E1 -3060.72,E2 -3060.72} C_VEL
LIN {X 0,Y 559.238,Z 421.446,A -85,B 0,C 180,E1 -3062.882,E2 -3062.882} C_VEL
LIN {X 0,Y 559.23,Z 421.445,A -85,B 0,C 180,E1 -3065.77,E2 -3065.77} C_VEL
LIN {X 0,Y 559.197,Z 421.454,A -85,B 0,C 180,E1 -3068.674,E2 -3068.674} C_VEL
LIN {X 0,Y 559.198,Z 421.448,A -85,B 0,C 180,E1 -3071.601,E2 -3071.601} C_VEL
LIN {X 0,Y 559.192,Z 421.456,A -85,B 0,C 180,E1 -3074.596,E2 -3074.596} C_VEL
LIN {X 0,Y 559.158,Z 421.454,A -85,B 0,C 180,E1 -3077.557,E2 -3077.557} C_VEL
LIN {X 0,Y 559.169,Z 421.454,A -85,B 0,C 180,E1 -3079.838,E2 -3079.838} C_VEL
LIN {X 0,Y 559.138,Z 421.461,A -85,B 0,C 180,E1 -3082.153,E2 -3082.153} C_VEL
LIN {X 0,Y 559.174,Z 421.453,A -85,B 0,C 180,E1 -3085.188,E2 -3085.188} C_VEL
LIN {X 0,Y 559.19,Z 421.451,A -85,B 0,C 180,E1 -3087.712,E2 -3087.712} C_VEL
LIN {X 0,Y 559.148,Z 421.457,A -85,B 0,C 180,E1 -3090.63,E2 -3090.63} C_VEL
LIN {X 0,Y 558.485,Z 421.54,A -85,B 0,C 180,E1 -3091.231,E2 -3091.231} C_VEL
LIN {X 0,Y 555.622,Z 421.901,A -85,B 0,C 180,E1 -3092.207,E2 -3092.207} C_VEL
LIN {X 0,Y 553.211,Z 422.197,A -85,B 0,C 180,E1 -3092.993,E2 -3092.993} C_VEL
LIN {X 0,Y 552.193,Z 422.322,A -85,B 0,C 180,E1 -3093.6,E2 -3093.6} C_VEL
LIN {X 0,Y 552.119,Z 422.332,A -85,B 0,C 180,E1 -3093.805,E2 -3093.805} C_VEL
LIN {X 0,Y 552.113,Z 422.338,A -85,B 0,C 180,E1 -3096.747,E2 -3096.747} C_VEL
LIN {X 0,Y 552.132,Z 422.331,A -85,B 0,C 180,E1 -3099.527,E2 -3099.527} C_VEL
LIN {X 0,Y 552.127,Z 422.339,A -85,B 0,C 180,E1 -3102.426,E2 -3102.426} C_VEL
LIN {X 0,Y 552.139,Z 422.451,A -85,B 0,C 180,E1 -3104.179,E2 -3104.179} C_VEL
LIN {X 0,Y 553.462,Z 429.722,A -85,B 0,C 180,E1 -3105.325,E2 -3105.325} C_VEL
LIN {X 0,Y 553.115,Z 446.061,A -85,B 0,C 180,E1 -3107.678,E2 -3107.678} C_VEL
LIN {X 0,Y 555.165,Z 456.387,A -85,B 0,C 180,E1 -3107.896,E2 -3107.896} C_VEL
LIN {X 0,Y 554.495,Z 611.075,A -85,B 0,C 180,E1 -3109.968,E2 -3109.968} C_VEL
LIN {X 0,Y 554.251,Z 626.831,A -85,B 0,C 180,E1 -3110.331,E2 -3110.331} C_VEL
LIN {X 0,Y 553.972,Z 642.601,A -85,B 0,C 180,E1 -3110.866,E2 -3110.866} C_VEL
LIN {X 0,Y 553.737,Z 656.481,A -85,B 0,C 180,E1 -3111.488,E2 -3111.488} C_VEL
LIN {X 0,Y 553.389,Z 670.305,A -85,B 0,C 180,E1 -3112.264,E2 -3112.264} C_VEL
LIN {X 0,Y 553.056,Z 683.658,A -85,B 0,C 180,E1 -3113.186,E2 -3113.186} C_VEL
LIN {X 0,Y 552.77,Z 695.904,A -85,B 0,C 180,E1 -3114.209,E2 -3114.209} C_VEL
LIN {X 0,Y 552.447,Z 706.635,A -85,B 0,C 180,E1 -3115.275,E2 -3115.275} C_VEL
LIN {X 0,Y 552.251,Z 716.117,A -85,B 0,C 180,E1 -3116.388,E2 -3116.388} C_VEL
LIN {X 0,Y 552.071,Z 725.425,A -85,B 0,C 180,E1 -3117.679,E2 -3117.679} C_VEL
LIN {X 0,Y 551.918,Z 733.163,A -85,B 0,C 180,E1 -3118.965,E2 -3118.965} C_VEL
LIN {X 0,Y 551.841,Z 739.472,A -85,B 0,C 180,E1 -3120.22,E2 -3120.22} C_VEL
LIN {X 0,Y 551.75,Z 744.795,A -85,B 0,C 180,E1 -3121.51,E2 -3121.51} C_VEL
LIN {X 0,Y 551.725,Z 749.837,A -85,B 0,C 180,E1 -3123.085,E2 -3123.085} C_VEL
LIN {X 0,Y 551.659,Z 753.606,A -85,B 0,C 180,E1 -3124.76,E2 -3124.76} C_VEL
LIN {X 0,Y 551.655,Z 755.873,A -85,B 0,C 180,E1 -3126.531,E2 -3126.531} C_VEL
LIN {X 0,Y 551.615,Z 756.395,A -85,B 0,C 180,E1 -3127.529,E2 -3127.529} C_VEL
LIN {X 0,Y 551.643,Z 756.173,A -85,B 0,C 180,E1 -3129.102,E2 -3129.102} C_VEL
LIN {X 0,Y 551.684,Z 754.655,A -85,B 0,C 180,E1 -3130.658,E2 -3130.658} C_VEL
LIN {X 0,Y 551.67,Z 751.853,A -85,B 0,C 180,E1 -3132.197,E2 -3132.197} C_VEL
LIN {X 0,Y 551.755,Z 747.724,A -85,B 0,C 180,E1 -3133.727,E2 -3133.727} C_VEL
LIN {X 0,Y 551.834,Z 742.21,A -85,B 0,C 180,E1 -3135.244,E2 -3135.244} C_VEL
LIN {X 0,Y 551.906,Z 735.209,A -85,B 0,C 180,E1 -3136.75,E2 -3136.75} C_VEL
LIN {X 0,Y 552.076,Z 727.683,A -85,B 0,C 180,E1 -3138.062,E2 -3138.062} C_VEL
LIN {X 0,Y 552.209,Z 718.717,A -85,B 0,C 180,E1 -3139.366,E2 -3139.366} C_VEL
LIN {X 0,Y 552.399,Z 709.623,A -85,B 0,C 180,E1 -3140.48,E2 -3140.48} C_VEL
LIN {X 0,Y 552.68,Z 698.952,A -85,B 0,C 180,E1 -3141.592,E2 -3141.592} C_VEL
LIN {X 0,Y 552.996,Z 686.237,A -85,B 0,C 180,E1 -3142.699,E2 -3142.699} C_VEL
LIN {X 0,Y 553.279,Z 673.493,A -85,B 0,C 180,E1 -3143.619,E2 -3143.619} C_VEL
LIN {X 0,Y 553.654,Z 659.451,A -85,B 0,C 180,E1 -3144.446,E2 -3144.446} C_VEL
LIN {X 0,Y 553.947,Z 644.777,A -85,B 0,C 180,E1 -3145.133,E2 -3145.133} C_VEL
LIN {X 0,Y 554.219,Z 630.036,A -85,B 0,C 180,E1 -3145.66,E2 -3145.66} C_VEL
LIN {X 0,Y 554.386,Z 614.842,A -85,B 0,C 180,E1 -3146.048,E2 -3146.048} C_VEL
LIN {X 0,Y 554.551,Z 594.054,A -85,B 0,C 180,E1 -3146.367,E2 -3146.367} C_VEL
LIN {X 0,Y 555.155,Z 455.597,A -85,B 0,C 180,E1 -3148.205,E2 -3148.205} C_VEL
LIN {X 0,Y 553.115,Z 445.871,A -85,B 0,C 180,E1 -3148.424,E2 -3148.424} C_VEL
LIN {X 0,Y 553.387,Z 428.748,A -85,B 0,C 180,E1 -3150.91,E2 -3150.91} C_VEL
LIN {X 0,Y 552.209,Z 422.328,A -85,B 0,C 180,E1 -3151.961,E2 -3151.961} C_VEL
LIN {X 0,Y 552.229,Z 422.322,A -85,B 0,C 180,E1 -3155.111,E2 -3155.111} C_VEL
LIN {X 0,Y 552.163,Z 422.33,A -85,B 0,C 180,E1 -3158.049,E2 -3158.049} C_VEL
LIN {X 0,Y 552.167,Z 422.324,A -85,B 0,C 180,E1 -3161.007,E2 -3161.007} C_VEL
LIN {X 0,Y 552.141,Z 422.333,A -85,B 0,C 180,E1 -3163.996,E2 -3163.996} C_VEL
LIN {X 0,Y 552.138,Z 422.33,A -85,B 0,C 180,E1 -3167.023,E2 -3167.023} C_VEL
LIN {X 0,Y 552.134,Z 422.331,A -85,B 0,C 180,E1 -3170.101,E2 -3170.101} C_VEL
LIN {X 0,Y 552.1,Z 422.334,A -85,B 0,C 180,E1 -3172.451,E2 -3172.451} C_VEL
LIN {X 0,Y 552.16,Z 422.329,A -85,B 0,C 180,E1 -3175.35,E2 -3175.35} C_VEL
LIN {X 0,Y 552.124,Z 422.331,A -85,B 0,C 180,E1 -3178.098,E2 -3178.098} C_VEL
LIN {X 0,Y 552.111,Z 422.331,A -85,B 0,C 180,E1 -3180.609,E2 -3180.609} C_VEL
LIN {X 0,Y 552.127,Z 422.329,A -85,B 0,C 180,E1 -3183.185,E2 -3183.185} C_VEL
LIN {X 0,Y 552.112,Z 422.337,A -85,B 0,C 180,E1 -3185.842,E2 -3185.842} C_VEL
LIN {X 0,Y 552.129,Z 422.328,A -85,B 0,C 180,E1 -3189.062,E2 -3189.062} C_VEL
LIN {X 0,Y 552.143,Z 422.334,A -85,B 0,C 180,E1 -3191.444,E2 -3191.444} C_VEL
LIN {X 0,Y 552.099,Z 422.332,A -85,B 0,C 180,E1 -3194.532,E2 -3194.532} C_VEL
LIN {X 0,Y 552.133,Z 422.337,A -85,B 0,C 180,E1 -3197.584,E2 -3197.584} C_VEL
LIN {X 0,Y 552.136,Z 422.328,A -85,B 0,C 180,E1 -3200.473,E2 -3200.473} C_VEL
LIN {X 0,Y 552.124,Z 422.333,A -85,B 0,C 180,E1 -3203.314,E2 -3203.314} C_VEL
LIN {X 0,Y 552.133,Z 422.334,A -85,B 0,C 180,E1 -3205.939,E2 -3205.939} C_VEL
LIN {X 0,Y 552.12,Z 422.329,A -85,B 0,C 180,E1 -3208.54,E2 -3208.54} C_VEL
LIN {X 0,Y 552.127,Z 422.333,A -85,B 0,C 180,E1 -3211.437,E2 -3211.437} C_VEL
LIN {X 0,Y 552.138,Z 422.328,A -85,B 0,C 180,E1 -3214.356,E2 -3214.356} C_VEL
LIN {X 0,Y 552.099,Z 422.329,A -85,B 0,C 180,E1 -3216.758,E2 -3216.758} C_VEL
LIN {X 0,Y 552.121,Z 422.331,A -85,B 0,C 180,E1 -3219.12,E2 -3219.12} C_VEL
LIN {X 0,Y 552.127,Z 422.335,A -85,B 0,C 180,E1 -3221.444,E2 -3221.444} C_VEL
LIN {X 0,Y 552.12,Z 422.336,A -85,B 0,C 180,E1 -3223.737,E2 -3223.737} C_VEL
LIN {X 0,Y 552.136,Z 422.333,A -85,B 0,C 180,E1 -3226.004,E2 -3226.004} C_VEL
LIN {X 0,Y 552.163,Z 422.324,A -85,B 0,C 180,E1 -3228.993,E2 -3228.993} C_VEL
LIN {X 0,Y 552.16,Z 422.33,A -85,B 0,C 180,E1 -3231.951,E2 -3231.951} C_VEL
LIN {X 0,Y 552.23,Z 422.316,A -85,B 0,C 180,E1 -3234.889,E2 -3234.889} C_VEL
LIN {X 0,Y 552.223,Z 422.324,A -85,B 0,C 180,E1 -3237.812,E2 -3237.812} C_VEL
LIN {X 0,Y 552.243,Z 422.315,A -85,B 0,C 180,E1 -3240.729,E2 -3240.729} C_VEL
LIN {X 0,Y 552.207,Z 422.318,A -85,B 0,C 180,E1 -3242.918,E2 -3242.918} C_VEL
LIN {X 0,Y 552.198,Z 422.327,A -85,B 0,C 180,E1 -3245.844,E2 -3245.844} C_VEL
LIN {X 0,Y 552.162,Z 422.325,A -85,B 0,C 180,E1 -3248.785,E2 -3248.785} C_VEL
LIN {X 0,Y 552.162,Z 422.33,A -85,B 0,C 180,E1 -3251.75,E2 -3251.75} C_VEL
LIN {X 0,Y 552.136,Z 422.328,A -85,B 0,C 180,E1 -3254.748,E2 -3254.748} C_VEL
LIN {X 0,Y 552.11,Z 422.336,A -85,B 0,C 180,E1 -3257.788,E2 -3257.788} C_VEL
LIN {X 0,Y 552.13,Z 422.332,A -85,B 0,C 180,E1 -3260.101,E2 -3260.101} C_VEL
LIN {X 0,Y 552.095,Z 422.333,A -85,B 0,C 180,E1 -3262.451,E2 -3262.451} C_VEL
LIN {X 0,Y 552.155,Z 422.33,A -85,B 0,C 180,E1 -3265.35,E2 -3265.35} C_VEL
LIN {X 0,Y 552.125,Z 422.333,A -85,B 0,C 180,E1 -3268.097,E2 -3268.097} C_VEL
LIN {X 0,Y 552.101,Z 422.332,A -85,B 0,C 180,E1 -3270.609,E2 -3270.609} C_VEL
LIN {X 0,Y 552.122,Z 422.332,A -85,B 0,C 180,E1 -3273.185,E2 -3273.185} C_VEL
LIN {X 0,Y 552.113,Z 422.339,A -85,B 0,C 180,E1 -3275.841,E2 -3275.841} C_VEL
LIN {X 0,Y 552.124,Z 422.331,A -85,B 0,C 180,E1 -3279.062,E2 -3279.062} C_VEL
LIN {X 0,Y 552.127,Z 422.335,A -85,B 0,C 180,E1 -3281.445,E2 -3281.445} C_VEL
LIN {X 0,Y 552.095,Z 422.334,A -85,B 0,C 180,E1 -3284.532,E2 -3284.532} C_VEL
LIN {X 0,Y 552.131,Z 422.337,A -85,B 0,C 180,E1 -3287.584,E2 -3287.584} C_VEL
LIN {X 0,Y 552.131,Z 422.33,A -85,B 0,C 180,E1 -3290.473,E2 -3290.473} C_VEL
LIN {X 0,Y 552.106,Z 422.336,A -85,B 0,C 180,E1 -3293.317,E2 -3293.317} C_VEL
LIN {X 0,Y 552.127,Z 422.338,A -85,B 0,C 180,E1 -3295.939,E2 -3295.939} C_VEL
LIN {X 0,Y 552.12,Z 422.333,A -85,B 0,C 180,E1 -3298.541,E2 -3298.541} C_VEL
LIN {X 0,Y 552.125,Z 422.339,A -85,B 0,C 180,E1 -3301.438,E2 -3301.438} C_VEL
LIN {X 0,Y 552.133,Z 422.372,A -85,B 0,C 180,E1 -3302.925,E2 -3302.925} C_VEL
LIN {X 0,Y 554.198,Z 431.56,A -85,B 0,C 180,E1 -3304.208,E2 -3304.208} C_VEL
LIN {X 0,Y 553.761,Z 454.023,A -85,B 0,C 180,E1 -3307.029,E2 -3307.029} C_VEL
LIN {X 0,Y 553.372,Z 474.87,A -85,B 0,C 180,E1 -3309.621,E2 -3309.621} C_VEL
LIN {X 0,Y 555.159,Z 485.033,A -85,B 0,C 180,E1 -3309.832,E2 -3309.832} C_VEL
LIN {X 0,Y 554.469,Z 641.105,A -85,B 0,C 180,E1 -3311.922,E2 -3311.922} C_VEL
LIN {X 0,Y 554.295,Z 656.696,A -85,B 0,C 180,E1 -3312.284,E2 -3312.284} C_VEL
LIN {X 0,Y 554.036,Z 672.031,A -85,B 0,C 180,E1 -3312.799,E2 -3312.799} C_VEL
LIN {X 0,Y 553.795,Z 685.772,A -85,B 0,C 180,E1 -3313.409,E2 -3313.409} C_VEL
LIN {X 0,Y 553.405,Z 699.246,A -85,B 0,C 180,E1 -3314.155,E2 -3314.155} C_VEL
LIN {X 0,Y 553.084,Z 712.298,A -85,B 0,C 180,E1 -3315.041,E2 -3315.041} C_VEL
LIN {X 0,Y 552.781,Z 724.29,A -85,B 0,C 180,E1 -3316.021,E2 -3316.021} C_VEL
LIN {X 0,Y 552.53,Z 735.747,A -85,B 0,C 180,E1 -3317.138,E2 -3317.138} C_VEL
LIN {X 0,Y 552.253,Z 746.435,A -85,B 0,C 180,E1 -3318.383,E2 -3318.383} C_VEL
LIN {X 0,Y 552.124,Z 754.854,A -85,B 0,C 180,E1 -3319.549,E2 -3319.549} C_VEL
LIN {X 0,Y 551.959,Z 762.733,A -85,B 0,C 180,E1 -3320.842,E2 -3320.842} C_VEL
LIN {X 0,Y 551.838,Z 770.089,A -85,B 0,C 180,E1 -3322.315,E2 -3322.315} C_VEL
LIN {X 0,Y 551.745,Z 775.646,A -85,B 0,C 180,E1 -3323.703,E2 -3323.703} C_VEL
LIN {X 0,Y 551.713,Z 779.385,A -85,B 0,C 180,E1 -3324.884,E2 -3324.884} C_VEL
LIN {X 0,Y 551.73,Z 782.888,A -85,B 0,C 180,E1 -3326.348,E2 -3326.348} C_VEL
LIN {X 0,Y 551.653,Z 785.191,A -85,B 0,C 180,E1 -3327.809,E2 -3327.809} C_VEL
LIN {X 0,Y 551.639,Z 786.348,A -85,B 0,C 180,E1 -3329.27,E2 -3329.27} C_VEL
LIN {X 0,Y 551.639,Z 786.348,A -85,B 0,C 180,E1 -3330.73,E2 -3330.73} C_VEL
LIN {X 0,Y 551.653,Z 785.189,A -85,B 0,C 180,E1 -3332.19,E2 -3332.19} C_VEL
LIN {X 0,Y 551.73,Z 782.887,A -85,B 0,C 180,E1 -3333.651,E2 -3333.651} C_VEL
LIN {X 0,Y 551.713,Z 779.388,A -85,B 0,C 180,E1 -3335.115,E2 -3335.115} C_VEL
LIN {X 0,Y 551.779,Z 774.611,A -85,B 0,C 180,E1 -3336.582,E2 -3336.582} C_VEL
LIN {X 0,Y 551.876,Z 768.424,A -85,B 0,C 180,E1 -3338.052,E2 -3338.052} C_VEL
LIN {X 0,Y 551.951,Z 760.649,A -85,B 0,C 180,E1 -3339.527,E2 -3339.527} C_VEL
LIN {X 0,Y 552.183,Z 752.372,A -85,B 0,C 180,E1 -3340.82,E2 -3340.82} C_VEL
LIN {X 0,Y 552.351,Z 742.396,A -85,B 0,C 180,E1 -3342.118,E2 -3342.118} C_VEL
LIN {X 0,Y 552.608,Z 732.192,A -85,B 0,C 180,E1 -3343.233,E2 -3343.233} C_VEL
LIN {X 0,Y 552.906,Z 720.026,A -85,B 0,C 180,E1 -3344.351,E2 -3344.351} C_VEL
LIN {X 0,Y 553.246,Z 707.452,A -85,B 0,C 180,E1 -3345.309,E2 -3345.309} C_VEL
LIN {X 0,Y 553.515,Z 694.519,A -85,B 0,C 180,E1 -3346.125,E2 -3346.125} C_VEL
LIN {X 0,Y 553.86,Z 679.839,A -85,B 0,C 180,E1 -3346.873,E2 -3346.873} C_VEL
LIN {X 0,Y 554.134,Z 665.631,A -85,B 0,C 180,E1 -3347.435,E2 -3347.435} C_VEL
LIN {X 0,Y 554.397,Z 650.533,A -85,B 0,C 180,E1 -3347.875,E2 -3347.875} C_VEL
LIN {X 0,Y 554.503,Z 636.343,A -85,B 0,C 180,E1 -3348.153,E2 -3348.153} C_VEL
LIN {X 0,Y 555.166,Z 484.431,A -85,B 0,C 180,E1 -3350.175,E2 -3350.175} C_VEL
LIN {X 0,Y 553.345,Z 474.827,A -85,B 0,C 180,E1 -3350.385,E2 -3350.385} C_VEL
LIN {X 0,Y 553.816,Z 450.864,A -85,B 0,C 180,E1 -3353.363,E2 -3353.363} C_VEL
LIN {X 0,Y 554.167,Z 431.565,A -85,B 0,C 180,E1 -3355.786,E2 -3355.786} C_VEL
LIN {X 0,Y 552.136,Z 422.337,A -85,B 0,C 180,E1 -3357.098,E2 -3357.098} C_VEL
LIN {X 0,Y 552.126,Z 422.339,A -85,B 0,C 180,E1 -3360.052,E2 -3360.052} C_VEL
LIN {X 0,Y 552.126,Z 422.332,A -85,B 0,C 180,E1 -3362.848,E2 -3362.848} C_VEL
LIN {X 0,Y 552.091,Z 422.334,A -85,B 0,C 180,E1 -3365.442,E2 -3365.442} C_VEL
LIN {X 0,Y 552.095,Z 422.337,A -85,B 0,C 180,E1 -3367.886,E2 -3367.886} C_VEL
LIN {X 0,Y 552.138,Z 422.336,A -85,B 0,C 180,E1 -3370.477,E2 -3370.477} C_VEL
LIN {X 0,Y 552.112,Z 422.331,A -85,B 0,C 180,E1 -3373.484,E2 -3373.484} C_VEL
LIN {X 0,Y 552.102,Z 422.337,A -85,B 0,C 180,E1 -3376.576,E2 -3376.576} C_VEL
LIN {X 0,Y 552.116,Z 422.331,A -85,B 0,C 180,E1 -3379.52,E2 -3379.52} C_VEL
LIN {X 0,Y 552.088,Z 422.343,A -85,B 0,C 180,E1 -3382.336,E2 -3382.336} C_VEL
LIN {X 0,Y 552.125,Z 422.33,A -85,B 0,C 180,E1 -3385.054,E2 -3385.054} C_VEL
LIN {X 0,Y 552.121,Z 422.331,A -85,B 0,C 180,E1 -3387.682,E2 -3387.682} C_VEL
LIN {X 0,Y 552.106,Z 422.34,A -85,B 0,C 180,E1 -3390.235,E2 -3390.235} C_VEL
LIN {X 0,Y 552.14,Z 422.328,A -85,B 0,C 180,E1 -3392.998,E2 -3392.998} C_VEL
LIN {X 0,Y 552.106,Z 422.332,A -85,B 0,C 180,E1 -3395.161,E2 -3395.161} C_VEL
LIN {X 0,Y 552.089,Z 422.334,A -85,B 0,C 180,E1 -3397.549,E2 -3397.549} C_VEL
LIN {X 0,Y 552.142,Z 422.336,A -85,B 0,C 180,E1 -3400.373,E2 -3400.373} C_VEL
LIN {X 0,Y 552.15,Z 422.326,A -85,B 0,C 180,E1 -3402.977,E2 -3402.977} C_VEL
LIN {X 0,Y 552.129,Z 422.333,A -85,B 0,C 180,E1 -3406.004,E2 -3406.004} C_VEL
LIN {X 0,Y 552.156,Z 422.327,A -85,B 0,C 180,E1 -3408.993,E2 -3408.993} C_VEL
LIN {X 0,Y 552.156,Z 422.329,A -85,B 0,C 180,E1 -3411.952,E2 -3411.952} C_VEL
LIN {X 0,Y 552.225,Z 422.319,A -85,B 0,C 180,E1 -3414.889,E2 -3414.889} C_VEL
LIN {X 0,Y 552.218,Z 422.319,A -85,B 0,C 180,E1 -3417.812,E2 -3417.812} C_VEL
LIN {X 0,Y 552.239,Z 422.318,A -85,B 0,C 180,E1 -3420.729,E2 -3420.729} C_VEL
LIN {X 0,Y 552.204,Z 422.322,A -85,B 0,C 180,E1 -3422.918,E2 -3422.918} C_VEL
LIN {X 0,Y 552.2,Z 422.322,A -85,B 0,C 180,E1 -3425.844,E2 -3425.844} C_VEL
LIN {X 0,Y 552.164,Z 422.329,A -85,B 0,C 180,E1 -3428.786,E2 -3428.786} C_VEL
LIN {X 0,Y 552.156,Z 422.326,A -85,B 0,C 180,E1 -3431.751,E2 -3431.751} C_VEL
LIN {X 0,Y 552.13,Z 422.334,A -85,B 0,C 180,E1 -3434.749,E2 -3434.749} C_VEL
LIN {X 0,Y 552.11,Z 422.333,A -85,B 0,C 180,E1 -3437.789,E2 -3437.789} C_VEL
LIN {X 0,Y 552.129,Z 422.334,A -85,B 0,C 180,E1 -3440.102,E2 -3440.102} C_VEL
LIN {X 0,Y 552.092,Z 422.344,A -85,B 0,C 180,E1 -3442.451,E2 -3442.451} C_VEL
LIN {X 0,Y 552.152,Z 422.327,A -85,B 0,C 180,E1 -3445.352,E2 -3445.352} C_VEL
LIN {X 0,Y 552.123,Z 422.335,A -85,B 0,C 180,E1 -3448.098,E2 -3448.098} C_VEL
LIN {X 0,Y 552.109,Z 422.339,A -85,B 0,C 180,E1 -3450.625,E2 -3450.625} C_VEL
LIN {X 0,Y 552.125,Z 422.331,A -85,B 0,C 180,E1 -3453.185,E2 -3453.185} C_VEL
LIN {X 0,Y 552.119,Z 422.332,A -85,B 0,C 180,E1 -3453.805,E2 -3453.805} C_VEL
LIN {X 0,Y 551.486,Z 422.418,A -85,B 0,C 180,E1 -3454.414,E2 -3454.414} C_VEL
LIN {X 0,Y 548.663,Z 422.772,A -85,B 0,C 180,E1 -3455.402,E2 -3455.402} C_VEL
LIN {X 0,Y 546.239,Z 423.072,A -85,B 0,C 180,E1 -3456.197,E2 -3456.197} C_VEL
LIN {X 0,Y 545.167,Z 423.203,A -85,B 0,C 180,E1 -3456.811,E2 -3456.811} C_VEL
LIN {X 0,Y 545.064,Z 423.213,A -85,B 0,C 180,E1 -3457.019,E2 -3457.019} C_VEL
LIN {X 0,Y 545.09,Z 423.214,A -85,B 0,C 180,E1 -3460.141,E2 -3460.141} C_VEL
LIN {X 0,Y 545.075,Z 423.215,A -85,B 0,C 180,E1 -3463.107,E2 -3463.107} C_VEL
LIN {X 0,Y 545.126,Z 423.402,A -85,B 0,C 180,E1 -3463.968,E2 -3463.968} C_VEL
LIN {X 0,Y 546.465,Z 429.919,A -85,B 0,C 180,E1 -3465.02,E2 -3465.02} C_VEL
LIN {X 0,Y 546.214,Z 445.361,A -85,B 0,C 180,E1 -3467.309,E2 -3467.309} C_VEL
LIN {X 0,Y 546.223,Z 446.148,A -85,B 0,C 180,E1 -3467.41,E2 -3467.41} C_VEL
LIN {X 0,Y 548.511,Z 457.343,A -85,B 0,C 180,E1 -3467.654,E2 -3467.654} C_VEL
LIN {X 0,Y 547.762,Z 610.967,A -85,B 0,C 180,E1 -3469.736,E2 -3469.736} C_VEL
LIN {X 0,Y 547.531,Z 625.744,A -85,B 0,C 180,E1 -3470.076,E2 -3470.076} C_VEL
LIN {X 0,Y 547.24,Z 640.143,A -85,B 0,C 180,E1 -3470.551,E2 -3470.551} C_VEL
LIN {X 0,Y 546.944,Z 654.429,A -85,B 0,C 180,E1 -3471.175,E2 -3471.175} C_VEL
LIN {X 0,Y 546.604,Z 667.511,A -85,B 0,C 180,E1 -3471.892,E2 -3471.892} C_VEL
LIN {X 0,Y 546.219,Z 680.931,A -85,B 0,C 180,E1 -3472.791,E2 -3472.791} C_VEL
LIN {X 0,Y 545.865,Z 693.784,A -85,B 0,C 180,E1 -3473.84,E2 -3473.84} C_VEL
LIN {X 0,Y 545.542,Z 704.746,A -85,B 0,C 180,E1 -3474.909,E2 -3474.909} C_VEL
LIN {X 0,Y 545.282,Z 715.216,A -85,B 0,C 180,E1 -3476.122,E2 -3476.122} C_VEL
LIN {X 0,Y 545.066,Z 724.684,A -85,B 0,C 180,E1 -3477.432,E2 -3477.432} C_VEL
LIN {X 0,Y 544.882,Z 732.051,A -85,B 0,C 180,E1 -3478.641,E2 -3478.641} C_VEL
LIN {X 0,Y 544.798,Z 738.023,A -85,B 0,C 180,E1 -3479.805,E2 -3479.805} C_VEL
LIN {X 0,Y 544.679,Z 744.437,A -85,B 0,C 180,E1 -3481.331,E2 -3481.331} C_VEL
LIN {X 0,Y 544.654,Z 749.544,A -85,B 0,C 180,E1 -3482.918,E2 -3482.918} C_VEL
LIN {X 0,Y 544.586,Z 752.159,A -85,B 0,C 180,E1 -3483.975,E2 -3483.975} C_VEL
LIN {X 0,Y 544.546,Z 754.95,A -85,B 0,C 180,E1 -3485.608,E2 -3485.608} C_VEL
LIN {X 0,Y 544.525,Z 756.323,A -85,B 0,C 180,E1 -3487.22,E2 -3487.22} C_VEL
LIN {X 0,Y 544.56,Z 756.341,A -85,B 0,C 180,E1 -3488.817,E2 -3488.817} C_VEL
LIN {X 0,Y 544.584,Z 755.038,A -85,B 0,C 180,E1 -3490.405,E2 -3490.405} C_VEL
LIN {X 0,Y 544.56,Z 752.472,A -85,B 0,C 180,E1 -3491.957,E2 -3491.957} C_VEL
LIN {X 0,Y 544.654,Z 748.579,A -85,B 0,C 180,E1 -3493.509,E2 -3493.509} C_VEL
LIN {X 0,Y 544.748,Z 743.326,A -85,B 0,C 180,E1 -3495.048,E2 -3495.048} C_VEL
LIN {X 0,Y 544.804,Z 736.628,A -85,B 0,C 180,E1 -3496.574,E2 -3496.574} C_VEL
LIN {X 0,Y 544.95,Z 729.417,A -85,B 0,C 180,E1 -3497.903,E2 -3497.903} C_VEL
LIN {X 0,Y 545.141,Z 720.79,A -85,B 0,C 180,E1 -3499.227,E2 -3499.227} C_VEL
LIN {X 0,Y 545.397,Z 710.47,A -85,B 0,C 180,E1 -3500.544,E2 -3500.544} C_VEL
LIN {X 0,Y 545.698,Z 699.964,A -85,B 0,C 180,E1 -3501.67,E2 -3501.67} C_VEL
LIN {X 0,Y 546.001,Z 689.137,A -85,B 0,C 180,E1 -3502.655,E2 -3502.655} C_VEL
LIN {X 0,Y 546.337,Z 676.339,A -85,B 0,C 180,E1 -3503.63,E2 -3503.63} C_VEL
LIN {X 0,Y 546.72,Z 662.974,A -85,B 0,C 180,E1 -3504.468,E2 -3504.468} C_VEL
LIN {X 0,Y 547.057,Z 648.17,A -85,B 0,C 180,E1 -3505.21,E2 -3505.21} C_VEL
LIN {X 0,Y 547.374,Z 633.114,A -85,B 0,C 180,E1 -3505.79,E2 -3505.79} C_VEL
LIN {X 0,Y 547.637,Z 618.193,A -85,B 0,C 180,E1 -3506.206,E2 -3506.206} C_VEL
LIN {X 0,Y 547.775,Z 602.821,A -85,B 0,C 180,E1 -3506.483,E2 -3506.483} C_VEL
LIN {X 0,Y 548.494,Z 456.902,A -85,B 0,C 180,E1 -3508.443,E2 -3508.443} C_VEL
LIN {X 0,Y 546.218,Z 445.989,A -85,B 0,C 180,E1 -3508.687,E2 -3508.687} C_VEL
LIN {X 0,Y 546.558,Z 430.854,A -85,B 0,C 180,E1 -3510.921,E2 -3510.921} C_VEL
LIN {X 0,Y 545.182,Z 423.202,A -85,B 0,C 180,E1 -3512.171,E2 -3512.171} C_VEL
LIN {X 0,Y 545.204,Z 423.197,A -85,B 0,C 180,E1 -3515.177,E2 -3515.177} C_VEL
LIN {X 0,Y 545.133,Z 423.205,A -85,B 0,C 180,E1 -3518.153,E2 -3518.153} C_VEL
LIN {X 0,Y 545.141,Z 423.205,A -85,B 0,C 180,E1 -3521.535,E2 -3521.535} C_VEL
LIN {X 0,Y 545.108,Z 423.205,A -85,B 0,C 180,E1 -3524.767,E2 -3524.767} C_VEL
LIN {X 0,Y 545.081,Z 423.211,A -85,B 0,C 180,E1 -3528.026,E2 -3528.026} C_VEL
LIN {X 0,Y 545.099,Z 423.205,A -85,B 0,C 180,E1 -3530.372,E2 -3530.372} C_VEL
LIN {X 0,Y 545.096,Z 423.214,A -85,B 0,C 180,E1 -3533.559,E2 -3533.559} C_VEL
LIN {X 0,Y 545.084,Z 423.211,A -85,B 0,C 180,E1 -3536,E2 -3536} C_VEL
LIN {X 0,Y 545.093,Z 423.204,A -85,B 0,C 180,E1 -3538.748,E2 -3538.748} C_VEL
LIN {X 0,Y 545.082,Z 423.213,A -85,B 0,C 180,E1 -3541.682,E2 -3541.682} C_VEL
LIN {X 0,Y 545.08,Z 423.207,A -85,B 0,C 180,E1 -3544.563,E2 -3544.563} C_VEL
LIN {X 0,Y 545.043,Z 423.215,A -85,B 0,C 180,E1 -3547.303,E2 -3547.303} C_VEL
LIN {X 0,Y 545.078,Z 423.21,A -85,B 0,C 180,E1 -3550.142,E2 -3550.142} C_VEL
LIN {X 0,Y 545.089,Z 423.206,A -85,B 0,C 180,E1 -3553.105,E2 -3553.105} C_VEL
LIN {X 0,Y 545.069,Z 423.21,A -85,B 0,C 180,E1 -3556.224,E2 -3556.224} C_VEL
LIN {X 0,Y 545.102,Z 423.202,A -85,B 0,C 180,E1 -3558.887,E2 -3558.887} C_VEL
LIN {X 0,Y 545.056,Z 423.217,A -85,B 0,C 180,E1 -3561.763,E2 -3561.763} C_VEL
LIN {X 0,Y 545.066,Z 423.207,A -85,B 0,C 180,E1 -3564.533,E2 -3564.533} C_VEL
LIN {X 0,Y 545.083,Z 423.21,A -85,B 0,C 180,E1 -3567.212,E2 -3567.212} C_VEL
LIN {X 0,Y 545.065,Z 423.214,A -85,B 0,C 180,E1 -3569.81,E2 -3569.81} C_VEL
LIN {X 0,Y 545.097,Z 423.206,A -85,B 0,C 180,E1 -3572.344,E2 -3572.344} C_VEL
LIN {X 0,Y 545.119,Z 423.202,A -85,B 0,C 180,E1 -3574.82,E2 -3574.82} C_VEL
LIN {X 0,Y 545.039,Z 423.211,A -85,B 0,C 180,E1 -3577.242,E2 -3577.242} C_VEL
LIN {X 0,Y 545.121,Z 423.202,A -85,B 0,C 180,E1 -3580.415,E2 -3580.415} C_VEL
LIN {X 0,Y 545.076,Z 423.212,A -85,B 0,C 180,E1 -3583.521,E2 -3583.521} C_VEL
LIN {X 0,Y 545.095,Z 423.212,A -85,B 0,C 180,E1 -3585.82,E2 -3585.82} C_VEL
LIN {X 0,Y 545.118,Z 423.201,A -85,B 0,C 180,E1 -3588.849,E2 -3588.849} C_VEL
LIN {X 0,Y 545.13,Z 423.207,A -85,B 0,C 180,E1 -3591.847,E2 -3591.847} C_VEL
LIN {X 0,Y 545.205,Z 423.191,A -85,B 0,C 180,E1 -3594.823,E2 -3594.823} C_VEL
LIN {X 0,Y 545.195,Z 423.199,A -85,B 0,C 180,E1 -3597.783,E2 -3597.783} C_VEL
LIN {X 0,Y 545.213,Z 423.19,A -85,B 0,C 180,E1 -3600.738,E2 -3600.738} C_VEL
LIN {X 0,Y 545.174,Z 423.194,A -85,B 0,C 180,E1 -3602.956,E2 -3602.956} C_VEL
LIN {X 0,Y 545.17,Z 423.201,A -85,B 0,C 180,E1 -3605.919,E2 -3605.919} C_VEL
LIN {X 0,Y 545.121,Z 423.202,A -85,B 0,C 180,E1 -3608.9,E2 -3608.9} C_VEL
LIN {X 0,Y 545.134,Z 423.203,A -85,B 0,C 180,E1 -3611.904,E2 -3611.904} C_VEL
LIN {X 0,Y 545.085,Z 423.207,A -85,B 0,C 180,E1 -3614.943,E2 -3614.943} C_VEL
LIN {X 0,Y 545.078,Z 423.208,A -85,B 0,C 180,E1 -3618.026,E2 -3618.026} C_VEL
LIN {X 0,Y 545.094,Z 423.206,A -85,B 0,C 180,E1 -3620.372,E2 -3620.372} C_VEL
LIN {X 0,Y 545.09,Z 423.213,A -85,B 0,C 180,E1 -3623.559,E2 -3623.559} C_VEL
LIN {X 0,Y 545.079,Z 423.212,A -85,B 0,C 180,E1 -3626,E2 -3626} C_VEL
LIN {X 0,Y 545.089,Z 423.205,A -85,B 0,C 180,E1 -3628.748,E2 -3628.748} C_VEL
LIN {X 0,Y 545.058,Z 423.218,A -85,B 0,C 180,E1 -3631.679,E2 -3631.679} C_VEL
LIN {X 0,Y 545.081,Z 423.207,A -85,B 0,C 180,E1 -3634.563,E2 -3634.563} C_VEL
LIN {X 0,Y 545.039,Z 423.216,A -85,B 0,C 180,E1 -3637.304,E2 -3637.304} C_VEL
LIN {X 0,Y 545.071,Z 423.212,A -85,B 0,C 180,E1 -3640.142,E2 -3640.142} C_VEL
LIN {X 0,Y 545.078,Z 423.209,A -85,B 0,C 180,E1 -3643.107,E2 -3643.107} C_VEL
LIN {X 0,Y 545.065,Z 423.212,A -85,B 0,C 180,E1 -3646.224,E2 -3646.224} C_VEL
LIN {X 0,Y 545.088,Z 423.207,A -85,B 0,C 180,E1 -3648.886,E2 -3648.886} C_VEL
LIN {X 0,Y 545.054,Z 423.22,A -85,B 0,C 180,E1 -3651.763,E2 -3651.763} C_VEL
LIN {X 0,Y 545.036,Z 423.215,A -85,B 0,C 180,E1 -3654.532,E2 -3654.532} C_VEL
LIN {X 0,Y 545.07,Z 423.213,A -85,B 0,C 180,E1 -3657.212,E2 -3657.212} C_VEL
LIN {X 0,Y 545.066,Z 423.219,A -85,B 0,C 180,E1 -3659.811,E2 -3659.811} C_VEL
LIN {X 0,Y 545.112,Z 423.299,A -85,B 0,C 180,E1 -3662.693,E2 -3662.693} C_VEL
LIN {X 0,Y 547.392,Z 433.361,A -85,B 0,C 180,E1 -3664.117,E2 -3664.117} C_VEL
LIN {X 0,Y 546.883,Z 455.439,A -85,B 0,C 180,E1 -3666.924,E2 -3666.924} C_VEL
LIN {X 0,Y 546.469,Z 474.888,A -85,B 0,C 180,E1 -3669.357,E2 -3669.357} C_VEL
LIN {X 0,Y 548.495,Z 485.682,A -85,B 0,C 180,E1 -3669.585,E2 -3669.585} C_VEL
LIN {X 0,Y 547.735,Z 641.516,A -85,B 0,C 180,E1 -3671.7,E2 -3671.7} C_VEL
LIN {X 0,Y 547.544,Z 656.694,A -85,B 0,C 180,E1 -3672.058,E2 -3672.058} C_VEL
LIN {X 0,Y 547.249,Z 670.793,A -85,B 0,C 180,E1 -3672.531,E2 -3672.531} C_VEL
LIN {X 0,Y 546.981,Z 683.795,A -85,B 0,C 180,E1 -3673.1,E2 -3673.1} C_VEL
LIN {X 0,Y 546.565,Z 697.671,A -85,B 0,C 180,E1 -3673.855,E2 -3673.855} C_VEL
LIN {X 0,Y 546.288,Z 709.61,A -85,B 0,C 180,E1 -3674.651,E2 -3674.651} C_VEL
LIN {X 0,Y 545.953,Z 722.151,A -85,B 0,C 180,E1 -3675.652,E2 -3675.652} C_VEL
LIN {X 0,Y 545.639,Z 732.182,A -85,B 0,C 180,E1 -3676.594,E2 -3676.594} C_VEL
LIN {X 0,Y 545.358,Z 742.389,A -85,B 0,C 180,E1 -3677.723,E2 -3677.723} C_VEL
LIN {X 0,Y 545.155,Z 752.366,A -85,B 0,C 180,E1 -3679.038,E2 -3679.038} C_VEL
LIN {X 0,Y 544.905,Z 760.647,A -85,B 0,C 180,E1 -3680.347,E2 -3680.347} C_VEL
LIN {X 0,Y 544.819,Z 768.422,A -85,B 0,C 180,E1 -3681.842,E2 -3681.842} C_VEL
LIN {X 0,Y 544.675,Z 775.18,A -85,B 0,C 180,E1 -3683.483,E2 -3683.483} C_VEL
LIN {X 0,Y 544.642,Z 779.386,A -85,B 0,C 180,E1 -3684.817,E2 -3684.817} C_VEL
LIN {X 0,Y 544.645,Z 782.888,A -85,B 0,C 180,E1 -3686.3,E2 -3686.3} C_VEL
LIN {X 0,Y 544.567,Z 785.19,A -85,B 0,C 180,E1 -3687.781,E2 -3687.781} C_VEL
LIN {X 0,Y 544.539,Z 786.348,A -85,B 0,C 180,E1 -3689.26,E2 -3689.26} C_VEL
LIN {X 0,Y 544.539,Z 786.348,A -85,B 0,C 180,E1 -3690.739,E2 -3690.739} C_VEL
LIN {X 0,Y 544.567,Z 785.188,A -85,B 0,C 180,E1 -3692.218,E2 -3692.218} C_VEL
LIN {X 0,Y 544.645,Z 782.886,A -85,B 0,C 180,E1 -3693.699,E2 -3693.699} C_VEL
LIN {X 0,Y 544.642,Z 779.388,A -85,B 0,C 180,E1 -3695.182,E2 -3695.182} C_VEL
LIN {X 0,Y 544.697,Z 774.611,A -85,B 0,C 180,E1 -3696.668,E2 -3696.668} C_VEL
LIN {X 0,Y 544.818,Z 768.423,A -85,B 0,C 180,E1 -3698.157,E2 -3698.157} C_VEL
LIN {X 0,Y 544.904,Z 760.648,A -85,B 0,C 180,E1 -3699.652,E2 -3699.652} C_VEL
LIN {X 0,Y 545.149,Z 752.371,A -85,B 0,C 180,E1 -3700.961,E2 -3700.961} C_VEL
LIN {X 0,Y 545.356,Z 742.396,A -85,B 0,C 180,E1 -3702.276,E2 -3702.276} C_VEL
LIN {X 0,Y 545.638,Z 732.191,A -85,B 0,C 180,E1 -3703.405,E2 -3703.405} C_VEL
LIN {X 0,Y 545.969,Z 720.026,A -85,B 0,C 180,E1 -3704.537,E2 -3704.537} C_VEL
LIN {X 0,Y 546.373,Z 706.387,A -85,B 0,C 180,E1 -3705.581,E2 -3705.581} C_VEL
LIN {X 0,Y 546.738,Z 692.889,A -85,B 0,C 180,E1 -3706.427,E2 -3706.427} C_VEL
LIN {X 0,Y 547.061,Z 678.814,A -85,B 0,C 180,E1 -3707.137,E2 -3707.137} C_VEL
LIN {X 0,Y 547.367,Z 664.323,A -85,B 0,C 180,E1 -3707.706,E2 -3707.706} C_VEL
LIN {X 0,Y 547.63,Z 648.965,A -85,B 0,C 180,E1 -3708.144,E2 -3708.144} C_VEL
LIN {X 0,Y 547.798,Z 633.716,A -85,B 0,C 180,E1 -3708.425,E2 -3708.425} C_VEL
LIN {X 0,Y 548.424,Z 484.599,A -85,B 0,C 180,E1 -3710.432,E2 -3710.432} C_VEL
LIN {X 0,Y 546.478,Z 474.808,A -85,B 0,C 180,E1 -3710.653,E2 -3710.653} C_VEL
LIN {X 0,Y 546.973,Z 450.808,A -85,B 0,C 180,E1 -3713.654,E2 -3713.654} C_VEL
LIN {X 0,Y 547.352,Z 433.265,A -85,B 0,C 180,E1 -3715.884,E2 -3715.884} C_VEL
LIN {X 0,Y 545.112,Z 423.213,A -85,B 0,C 180,E1 -3717.307,E2 -3717.307} C_VEL
LIN {X 0,Y 545.094,Z 423.215,A -85,B 0,C 180,E1 -3720.249,E2 -3720.249} C_VEL
LIN {X 0,Y 545.086,Z 423.208,A -85,B 0,C 180,E1 -3723.063,E2 -3723.063} C_VEL
LIN {X 0,Y 545.048,Z 423.213,A -85,B 0,C 180,E1 -3725.675,E2 -3725.675} C_VEL
LIN {X 0,Y 545.051,Z 423.219,A -85,B 0,C 180,E1 -3728.236,E2 -3728.236} C_VEL
LIN {X 0,Y 545.097,Z 423.206,A -85,B 0,C 180,E1 -3731.112,E2 -3731.112} C_VEL
LIN {X 0,Y 545.054,Z 423.216,A -85,B 0,C 180,E1 -3734.128,E2 -3734.128} C_VEL
LIN {X 0,Y 545.073,Z 423.209,A -85,B 0,C 180,E1 -3736.893,E2 -3736.893} C_VEL
LIN {X 0,Y 545.069,Z 423.212,A -85,B 0,C 180,E1 -3739.858,E2 -3739.858} C_VEL
LIN {X 0,Y 545.069,Z 423.21,A -85,B 0,C 180,E1 -3743.073,E2 -3743.073} C_VEL
LIN {X 0,Y 545.084,Z 423.208,A -85,B 0,C 180,E1 -3745.605,E2 -3745.605} C_VEL
LIN {X 0,Y 545.072,Z 423.218,A -85,B 0,C 180,E1 -3748.317,E2 -3748.317} C_VEL
LIN {X 0,Y 545.098,Z 423.205,A -85,B 0,C 180,E1 -3751.508,E2 -3751.508} C_VEL
LIN {X 0,Y 545.093,Z 423.213,A -85,B 0,C 180,E1 -3754.49,E2 -3754.49} C_VEL
LIN {X 0,Y 545.037,Z 423.212,A -85,B 0,C 180,E1 -3757.242,E2 -3757.242} C_VEL
LIN {X 0,Y 545.114,Z 423.212,A -85,B 0,C 180,E1 -3760.415,E2 -3760.415} C_VEL
LIN {X 0,Y 545.069,Z 423.207,A -85,B 0,C 180,E1 -3763.521,E2 -3763.521} C_VEL
LIN {X 0,Y 545.088,Z 423.208,A -85,B 0,C 180,E1 -3765.82,E2 -3765.82} C_VEL
LIN {X 0,Y 545.111,Z 423.206,A -85,B 0,C 180,E1 -3768.849,E2 -3768.849} C_VEL
LIN {X 0,Y 545.127,Z 423.203,A -85,B 0,C 180,E1 -3771.847,E2 -3771.847} C_VEL
LIN {X 0,Y 545.2,Z 423.195,A -85,B 0,C 180,E1 -3774.823,E2 -3774.823} C_VEL
LIN {X 0,Y 545.19,Z 423.194,A -85,B 0,C 180,E1 -3777.784,E2 -3777.784} C_VEL
LIN {X 0,Y 545.208,Z 423.193,A -85,B 0,C 180,E1 -3780.739,E2 -3780.739} C_VEL
LIN {X 0,Y 545.17,Z 423.198,A -85,B 0,C 180,E1 -3782.956,E2 -3782.956} C_VEL
LIN {X 0,Y 545.172,Z 423.198,A -85,B 0,C 180,E1 -3785.92,E2 -3785.92} C_VEL
LIN {X 0,Y 545.121,Z 423.205,A -85,B 0,C 180,E1 -3788.9,E2 -3788.9} C_VEL
LIN {X 0,Y 545.128,Z 423.203,A -85,B 0,C 180,E1 -3791.905,E2 -3791.905} C_VEL
LIN {X 0,Y 545.079,Z 423.21,A -85,B 0,C 180,E1 -3794.944,E2 -3794.944} C_VEL
LIN {X 0,Y 545.078,Z 423.211,A -85,B 0,C 180,E1 -3798.026,E2 -3798.026} C_VEL
LIN {X 0,Y 545.093,Z 423.215,A -85,B 0,C 180,E1 -3800.372,E2 -3800.372} C_VEL
LIN {X 0,Y 545.086,Z 423.207,A -85,B 0,C 180,E1 -3803.559,E2 -3803.559} C_VEL
LIN {X 0,Y 545.084,Z 423.211,A -85,B 0,C 180,E1 -3806.001,E2 -3806.001} C_VEL
LIN {X 0,Y 545.089,Z 423.211,A -85,B 0,C 180,E1 -3808.75,E2 -3808.75} C_VEL
LIN {X 0,Y 545.073,Z 423.21,A -85,B 0,C 180,E1 -3811.683,E2 -3811.683} C_VEL
LIN {X 0,Y 545.081,Z 423.214,A -85,B 0,C 180,E1 -3814.563,E2 -3814.563} C_VEL
LIN {X 0,Y 545.064,Z 423.213,A -85,B 0,C 180,E1 -3817.019,E2 -3817.019} C_VEL
LIN {X 0,Y 544.357,Z 423.3,A -85,B 0,C 180,E1 -3817.635,E2 -3817.635} C_VEL
LIN {X 0,Y 541.502,Z 423.661,A -85,B 0,C 180,E1 -3818.636,E2 -3818.636} C_VEL
LIN {X 0,Y 539.124,Z 423.954,A -85,B 0,C 180,E1 -3819.442,E2 -3819.442} C_VEL
LIN {X 0,Y 538.12,Z 424.081,A -85,B 0,C 180,E1 -3820.064,E2 -3820.064} C_VEL
LIN {X 0,Y 538.044,Z 424.087,A -85,B 0,C 180,E1 -3820.275,E2 -3820.275} C_VEL
LIN {X 0,Y 538.029,Z 424.092,A -85,B 0,C 180,E1 -3823.369,E2 -3823.369} C_VEL
LIN {X 0,Y 538.074,Z 424.194,A -85,B 0,C 180,E1 -3823.725,E2 -3823.725} C_VEL
LIN {X 0,Y 539.661,Z 432.012,A -85,B 0,C 180,E1 -3825.004,E2 -3825.004} C_VEL
LIN {X 0,Y 539.353,Z 446.189,A -85,B 0,C 180,E1 -3827.127,E2 -3827.127} C_VEL
LIN {X 0,Y 541.876,Z 458.681,A -85,B 0,C 180,E1 -3827.409,E2 -3827.409} C_VEL
LIN {X 0,Y 541.037,Z 610.878,A -85,B 0,C 180,E1 -3829.498,E2 -3829.498} C_VEL
LIN {X 0,Y 540.787,Z 625.868,A -85,B 0,C 180,E1 -3829.847,E2 -3829.847} C_VEL
LIN {X 0,Y 540.48,Z 639.259,A -85,B 0,C 180,E1 -3830.292,E2 -3830.292} C_VEL
LIN {X 0,Y 540.114,Z 653.939,A -85,B 0,C 180,E1 -3830.931,E2 -3830.931} C_VEL
LIN {X 0,Y 539.74,Z 667.426,A -85,B 0,C 180,E1 -3831.676,E2 -3831.676} C_VEL
LIN {X 0,Y 539.374,Z 679.534,A -85,B 0,C 180,E1 -3832.489,E2 -3832.489} C_VEL
LIN {X 0,Y 538.99,Z 691.917,A -85,B 0,C 180,E1 -3833.486,E2 -3833.486} C_VEL
LIN {X 0,Y 538.628,Z 703.659,A -85,B 0,C 180,E1 -3834.621,E2 -3834.621} C_VEL
LIN {X 0,Y 538.316,Z 714.312,A -85,B 0,C 180,E1 -3835.849,E2 -3835.849} C_VEL
LIN {X 0,Y 538.029,Z 723.93,A -85,B 0,C 180,E1 -3837.175,E2 -3837.175} C_VEL
LIN {X 0,Y 537.853,Z 731.904,A -85,B 0,C 180,E1 -3838.489,E2 -3838.489} C_VEL
LIN {X 0,Y 537.709,Z 739.052,A -85,B 0,C 180,E1 -3839.915,E2 -3839.915} C_VEL
LIN {X 0,Y 537.603,Z 744.087,A -85,B 0,C 180,E1 -3841.15,E2 -3841.15} C_VEL
LIN {X 0,Y 537.571,Z 749.318,A -85,B 0,C 180,E1 -3842.77,E2 -3842.77} C_VEL
LIN {X 0,Y 537.467,Z 753.194,A -85,B 0,C 180,E1 -3844.457,E2 -3844.457} C_VEL
LIN {X 0,Y 537.439,Z 755.495,A -85,B 0,C 180,E1 -3846.086,E2 -3846.086} C_VEL
LIN {X 0,Y 537.413,Z 756.437,A -85,B 0,C 180,E1 -3847.714,E2 -3847.714} C_VEL
LIN {X 0,Y 537.446,Z 756.049,A -85,B 0,C 180,E1 -3849.325,E2 -3849.325} C_VEL
LIN {X 0,Y 537.48,Z 754.369,A -85,B 0,C 180,E1 -3850.92,E2 -3850.92} C_VEL
LIN {X 0,Y 537.526,Z 751.059,A -85,B 0,C 180,E1 -3852.642,E2 -3852.642} C_VEL
LIN {X 0,Y 537.586,Z 747.104,A -85,B 0,C 180,E1 -3854.066,E2 -3854.066} C_VEL
LIN {X 0,Y 537.69,Z 741.42,A -85,B 0,C 180,E1 -3855.621,E2 -3855.621} C_VEL
LIN {X 0,Y 537.766,Z 734.238,A -85,B 0,C 180,E1 -3857.164,E2 -3857.164} C_VEL
LIN {X 0,Y 538.004,Z 726.967,A -85,B 0,C 180,E1 -3858.446,E2 -3858.446} C_VEL
LIN {X 0,Y 538.207,Z 717.389,A -85,B 0,C 180,E1 -3859.847,E2 -3859.847} C_VEL
LIN {X 0,Y 538.54,Z 706.365,A -85,B 0,C 180,E1 -3861.18,E2 -3861.18} C_VEL
LIN {X 0,Y 538.916,Z 694.648,A -85,B 0,C 180,E1 -3862.359,E2 -3862.359} C_VEL
LIN {X 0,Y 539.265,Z 682.805,A -85,B 0,C 180,E1 -3863.359,E2 -3863.359} C_VEL
LIN {X 0,Y 539.705,Z 669.276,A -85,B 0,C 180,E1 -3864.302,E2 -3864.302} C_VEL
LIN {X 0,Y 540.078,Z 656.085,A -85,B 0,C 180,E1 -3865.055,E2 -3865.055} C_VEL
LIN {X 0,Y 540.421,Z 641.578,A -85,B 0,C 180,E1 -3865.712,E2 -3865.712} C_VEL
LIN {X 0,Y 540.768,Z 626.427,A -85,B 0,C 180,E1 -3866.228,E2 -3866.228} C_VEL
LIN {X 0,Y 540.98,Z 611.65,A -85,B 0,C 180,E1 -3866.579,E2 -3866.579} C_VEL
LIN {X 0,Y 541.847,Z 457.854,A -85,B 0,C 180,E1 -3868.693,E2 -3868.693} C_VEL
LIN {X 0,Y 539.375,Z 446.185,A -85,B 0,C 180,E1 -3868.96,E2 -3868.96} C_VEL
LIN {X 0,Y 539.647,Z 431.761,A -85,B 0,C 180,E1 -3871.12,E2 -3871.12} C_VEL
LIN {X 0,Y 538.148,Z 424.077,A -85,B 0,C 180,E1 -3872.386,E2 -3872.386} C_VEL
LIN {X 0,Y 538.162,Z 424.074,A -85,B 0,C 180,E1 -3875.245,E2 -3875.245} C_VEL
LIN {X 0,Y 538.09,Z 424.081,A -85,B 0,C 180,E1 -3878.261,E2 -3878.261} C_VEL
LIN {X 0,Y 538.122,Z 424.08,A -85,B 0,C 180,E1 -3881.615,E2 -3881.615} C_VEL
LIN {X 0,Y 538.064,Z 424.083,A -85,B 0,C 180,E1 -3884.857,E2 -3884.857} C_VEL
LIN {X 0,Y 538.064,Z 424.09,A -85,B 0,C 180,E1 -3887.54,E2 -3887.54} C_VEL
LIN {X 0,Y 538.043,Z 424.084,A -85,B 0,C 180,E1 -3890.651,E2 -3890.651} C_VEL
LIN {X 0,Y 538.029,Z 424.09,A -85,B 0,C 180,E1 -3893.887,E2 -3893.887} C_VEL
LIN {X 0,Y 538.047,Z 424.084,A -85,B 0,C 180,E1 -3896.367,E2 -3896.367} C_VEL
LIN {X 0,Y 538.035,Z 424.084,A -85,B 0,C 180,E1 -3898.933,E2 -3898.933} C_VEL
LIN {X 0,Y 538.032,Z 424.088,A -85,B 0,C 180,E1 -3901.89,E2 -3901.89} C_VEL
LIN {X 0,Y 538.03,Z 424.086,A -85,B 0,C 180,E1 -3904.62,E2 -3904.62} C_VEL
LIN {X 0,Y 538.011,Z 424.09,A -85,B 0,C 180,E1 -3907.17,E2 -3907.17} C_VEL
LIN {X 0,Y 538.033,Z 424.093,A -85,B 0,C 180,E1 -3909.796,E2 -3909.796} C_VEL
LIN {X 0,Y 538.027,Z 424.084,A -85,B 0,C 180,E1 -3912.785,E2 -3912.785} C_VEL
LIN {X 0,Y 538.032,Z 424.09,A -85,B 0,C 180,E1 -3915.925,E2 -3915.925} C_VEL
LIN {X 0,Y 538.08,Z 424.08,A -85,B 0,C 180,E1 -3919.249,E2 -3919.249} C_VEL
LIN {X 0,Y 537.996,Z 424.091,A -85,B 0,C 180,E1 -3922.122,E2 -3922.122} C_VEL
LIN {X 0,Y 538.022,Z 424.084,A -85,B 0,C 180,E1 -3924.917,E2 -3924.917} C_VEL
LIN {X 0,Y 538.028,Z 424.095,A -85,B 0,C 180,E1 -3927.618,E2 -3927.618} C_VEL
LIN {X 0,Y 538.018,Z 424.085,A -85,B 0,C 180,E1 -3930.239,E2 -3930.239} C_VEL
LIN {X 0,Y 538.073,Z 424.08,A -85,B 0,C 180,E1 -3932.796,E2 -3932.796} C_VEL
LIN {X 0,Y 538.05,Z 424.086,A -85,B 0,C 180,E1 -3935.292,E2 -3935.292} C_VEL
LIN {X 0,Y 538.023,Z 424.085,A -85,B 0,C 180,E1 -3938.546,E2 -3938.546} C_VEL
LIN {X 0,Y 538.038,Z 424.085,A -85,B 0,C 180,E1 -3940.94,E2 -3940.94} C_VEL
LIN {X 0,Y 538.027,Z 424.086,A -85,B 0,C 180,E1 -3943.299,E2 -3943.299} C_VEL
LIN {X 0,Y 538.064,Z 424.088,A -85,B 0,C 180,E1 -3945.63,E2 -3945.63} C_VEL
LIN {X 0,Y 538.077,Z 424.078,A -85,B 0,C 180,E1 -3948.701,E2 -3948.701} C_VEL
LIN {X 0,Y 538.087,Z 424.085,A -85,B 0,C 180,E1 -3951.739,E2 -3951.739} C_VEL
LIN {X 0,Y 538.163,Z 424.068,A -85,B 0,C 180,E1 -3954.755,E2 -3954.755} C_VEL
LIN {X 0,Y 538.167,Z 424.074,A -85,B 0,C 180,E1 -3957.755,E2 -3957.755} C_VEL
LIN {X 0,Y 538.183,Z 424.066,A -85,B 0,C 180,E1 -3960.748,E2 -3960.748} C_VEL
LIN {X 0,Y 538.14,Z 424.071,A -85,B 0,C 180,E1 -3962.994,E2 -3962.994} C_VEL
LIN {X 0,Y 538.123,Z 424.077,A -85,B 0,C 180,E1 -3965.997,E2 -3965.997} C_VEL
LIN {X 0,Y 538.071,Z 424.081,A -85,B 0,C 180,E1 -3969.017,E2 -3969.017} C_VEL
LIN {X 0,Y 538.083,Z 424.079,A -85,B 0,C 180,E1 -3972.062,E2 -3972.062} C_VEL
LIN {X 0,Y 538.045,Z 424.085,A -85,B 0,C 180,E1 -3975.144,E2 -3975.144} C_VEL
LIN {X 0,Y 538.031,Z 424.083,A -85,B 0,C 180,E1 -3978.27,E2 -3978.27} C_VEL
LIN {X 0,Y 538.038,Z 424.084,A -85,B 0,C 180,E1 -3980.651,E2 -3980.651} C_VEL
LIN {X 0,Y 538.024,Z 424.093,A -85,B 0,C 180,E1 -3983.887,E2 -3983.887} C_VEL
LIN {X 0,Y 538.042,Z 424.085,A -85,B 0,C 180,E1 -3986.367,E2 -3986.367} C_VEL
LIN {X 0,Y 538.03,Z 424.085,A -85,B 0,C 180,E1 -3988.934,E2 -3988.934} C_VEL
LIN {X 0,Y 538.013,Z 424.094,A -85,B 0,C 180,E1 -3991.888,E2 -3991.888} C_VEL
LIN {X 0,Y 538.031,Z 424.085,A -85,B 0,C 180,E1 -3994.621,E2 -3994.621} C_VEL
LIN {X 0,Y 538.007,Z 424.09,A -85,B 0,C 180,E1 -3997.17,E2 -3997.17} C_VEL
LIN {X 0,Y 538.027,Z 424.094,A -85,B 0,C 180,E1 -3999.796,E2 -3999.796} C_VEL
LIN {X 0,Y 538.018,Z 424.087,A -85,B 0,C 180,E1 -4002.786,E2 -4002.786} C_VEL
LIN {X 0,Y 538.029,Z 424.092,A -85,B 0,C 180,E1 -4005.925,E2 -4005.925} C_VEL
LIN {X 0,Y 538.049,Z 424.086,A -85,B 0,C 180,E1 -4009.224,E2 -4009.224} C_VEL
LIN {X 0,Y 537.993,Z 424.094,A -85,B 0,C 180,E1 -4012.122,E2 -4012.122} C_VEL
LIN {X 0,Y 537.999,Z 424.092,A -85,B 0,C 180,E1 -4014.916,E2 -4014.916} C_VEL
LIN {X 0,Y 538.02,Z 424.095,A -85,B 0,C 180,E1 -4017.617,E2 -4017.617} C_VEL
LIN {X 0,Y 538.018,Z 424.094,A -85,B 0,C 180,E1 -4020.239,E2 -4020.239} C_VEL
LIN {X 0,Y 538.089,Z 424.236,A -85,B 0,C 180,E1 -4022.458,E2 -4022.458} C_VEL
LIN {X 0,Y 540.551,Z 434.899,A -85,B 0,C 180,E1 -4023.991,E2 -4023.991} C_VEL
LIN {X 0,Y 540.012,Z 456.838,A -85,B 0,C 180,E1 -4026.816,E2 -4026.816} C_VEL
LIN {X 0,Y 539.591,Z 474.713,A -85,B 0,C 180,E1 -4029.081,E2 -4029.081} C_VEL
LIN {X 0,Y 541.836,Z 486.413,A -85,B 0,C 180,E1 -4029.336,E2 -4029.336} C_VEL
LIN {X 0,Y 541.013,Z 640.919,A -85,B 0,C 180,E1 -4031.453,E2 -4031.453} C_VEL
LIN {X 0,Y 540.819,Z 656.197,A -85,B 0,C 180,E1 -4031.813,E2 -4031.813} C_VEL
LIN {X 0,Y 540.478,Z 670.793,A -85,B 0,C 180,E1 -4032.305,E2 -4032.305} C_VEL
LIN {X 0,Y 540.166,Z 683.793,A -85,B 0,C 180,E1 -4032.88,E2 -4032.88} C_VEL
LIN {X 0,Y 539.704,Z 697.669,A -85,B 0,C 180,E1 -4033.644,E2 -4033.644} C_VEL
LIN {X 0,Y 539.364,Z 710.494,A -85,B 0,C 180,E1 -4034.516,E2 -4034.516} C_VEL
LIN {X 0,Y 538.982,Z 723.218,A -85,B 0,C 180,E1 -4035.559,E2 -4035.559} C_VEL
LIN {X 0,Y 538.612,Z 733.963,A -85,B 0,C 180,E1 -4036.608,E2 -4036.608} C_VEL
LIN {X 0,Y 538.306,Z 743.901,A -85,B 0,C 180,E1 -4037.751,E2 -4037.751} C_VEL
LIN {X 0,Y 538.111,Z 753.621,A -85,B 0,C 180,E1 -4039.083,E2 -4039.083} C_VEL
LIN {X 0,Y 537.825,Z 761.723,A -85,B 0,C 180,E1 -4040.409,E2 -4040.409} C_VEL
LIN {X 0,Y 537.734,Z 768.422,A -85,B 0,C 180,E1 -4041.734,E2 -4041.734} C_VEL
LIN {X 0,Y 537.618,Z 774.604,A -85,B 0,C 180,E1 -4043.243,E2 -4043.243} C_VEL
LIN {X 0,Y 537.574,Z 779.385,A -85,B 0,C 180,E1 -4044.749,E2 -4044.749} C_VEL
LIN {X 0,Y 537.562,Z 782.887,A -85,B 0,C 180,E1 -4046.252,E2 -4046.252} C_VEL
LIN {X 0,Y 537.486,Z 785.19,A -85,B 0,C 180,E1 -4047.751,E2 -4047.751} C_VEL
LIN {X 0,Y 537.439,Z 786.348,A -85,B 0,C 180,E1 -4049.25,E2 -4049.25} C_VEL
LIN {X 0,Y 537.439,Z 786.347,A -85,B 0,C 180,E1 -4050.749,E2 -4050.749} C_VEL
LIN {X 0,Y 537.486,Z 785.187,A -85,B 0,C 180,E1 -4052.248,E2 -4052.248} C_VEL
LIN {X 0,Y 537.561,Z 782.885,A -85,B 0,C 180,E1 -4053.748,E2 -4053.748} C_VEL
LIN {X 0,Y 537.574,Z 779.388,A -85,B 0,C 180,E1 -4055.25,E2 -4055.25} C_VEL
LIN {X 0,Y 537.617,Z 774.611,A -85,B 0,C 180,E1 -4056.756,E2 -4056.756} C_VEL
LIN {X 0,Y 537.734,Z 768.423,A -85,B 0,C 180,E1 -4058.265,E2 -4058.265} C_VEL
LIN {X 0,Y 537.859,Z 760.647,A -85,B 0,C 180,E1 -4059.779,E2 -4059.779} C_VEL
LIN {X 0,Y 538.101,Z 752.371,A -85,B 0,C 180,E1 -4061.107,E2 -4061.107} C_VEL
LIN {X 0,Y 538.357,Z 742.396,A -85,B 0,C 180,E1 -4062.438,E2 -4062.438} C_VEL
LIN {X 0,Y 538.661,Z 732.19,A -85,B 0,C 180,E1 -4063.582,E2 -4063.582} C_VEL
LIN {X 0,Y 539.02,Z 720.025,A -85,B 0,C 180,E1 -4064.729,E2 -4064.729} C_VEL
LIN {X 0,Y 539.466,Z 707.834,A -85,B 0,C 180,E1 -4065.681,E2 -4065.681} C_VEL
LIN {X 0,Y 539.842,Z 694.514,A -85,B 0,C 180,E1 -4066.545,E2 -4066.545} C_VEL
LIN {X 0,Y 540.226,Z 679.834,A -85,B 0,C 180,E1 -4067.312,E2 -4067.312} C_VEL
LIN {X 0,Y 540.581,Z 664.323,A -85,B 0,C 180,E1 -4067.936,E2 -4067.936} C_VEL
LIN {X 0,Y 540.913,Z 648.765,A -85,B 0,C 180,E1 -4068.383,E2 -4068.383} C_VEL
LIN {X 0,Y 541.094,Z 633.233,A -85,B 0,C 180,E1 -4068.669,E2 -4068.669} C_VEL
LIN {X 0,Y 541.847,Z 486.43,A -85,B 0,C 180,E1 -4070.663,E2 -4070.663} C_VEL
LIN {X 0,Y 539.578,Z 474.602,A -85,B 0,C 180,E1 -4070.929,E2 -4070.929} C_VEL
LIN {X 0,Y 540.148,Z 450.839,A -85,B 0,C 180,E1 -4073.941,E2 -4073.941} C_VEL
LIN {X 0,Y 540.508,Z 434.818,A -85,B 0,C 180,E1 -4076.005,E2 -4076.005} C_VEL
LIN {X 0,Y 538.064,Z 424.093,A -85,B 0,C 180,E1 -4077.568,E2 -4077.568} C_VEL
LIN {X 0,Y 538.025,Z 424.093,A -85,B 0,C 180,E1 -4080.626,E2 -4080.626} C_VEL
LIN {X 0,Y 538.042,Z 424.086,A -85,B 0,C 180,E1 -4083.282,E2 -4083.282} C_VEL
LIN {X 0,Y 538.021,Z 424.092,A -85,B 0,C 180,E1 -4086.002,E2 -4086.002} C_VEL
LIN {X 0,Y 538.012,Z 424.09,A -85,B 0,C 180,E1 -4088.829,E2 -4088.829} C_VEL
LIN {X 0,Y 538.073,Z 424.084,A -85,B 0,C 180,E1 -4090.772,E2 -4090.772} C_VEL
LIN {X 0,Y 538.025,Z 424.091,A -85,B 0,C 180,E1 -4094.074,E2 -4094.074} C_VEL
LIN {X 0,Y 538.013,Z 424.087,A -85,B 0,C 180,E1 -4097.214,E2 -4097.214} C_VEL
LIN {X 0,Y 538.024,Z 424.094,A -85,B 0,C 180,E1 -4100.203,E2 -4100.203} C_VEL
LIN {X 0,Y 538.023,Z 424.087,A -85,B 0,C 180,E1 -4103.067,E2 -4103.067} C_VEL
LIN {X 0,Y 538.027,Z 424.089,A -85,B 0,C 180,E1 -4105.827,E2 -4105.827} C_VEL
LIN {X 0,Y 538.017,Z 424.094,A -85,B 0,C 180,E1 -4108.499,E2 -4108.499} C_VEL
LIN {X 0,Y 538.052,Z 424.083,A -85,B 0,C 180,E1 -4111.1,E2 -4111.1} C_VEL
LIN {X 0,Y 538.043,Z 424.084,A -85,B 0,C 180,E1 -4113.634,E2 -4113.634} C_VEL
LIN {X 0,Y 538.015,Z 424.093,A -85,B 0,C 180,E1 -4116.118,E2 -4116.118} C_VEL
LIN {X 0,Y 538.035,Z 424.083,A -85,B 0,C 180,E1 -4119.349,E2 -4119.349} C_VEL
LIN {X 0,Y 538.065,Z 424.086,A -85,B 0,C 180,E1 -4122.518,E2 -4122.518} C_VEL
LIN {X 0,Y 538.056,Z 424.083,A -85,B 0,C 180,E1 -4125.631,E2 -4125.631} C_VEL
LIN {X 0,Y 538.07,Z 424.085,A -85,B 0,C 180,E1 -4128.702,E2 -4128.702} C_VEL
LIN {X 0,Y 538.083,Z 424.08,A -85,B 0,C 180,E1 -4131.74,E2 -4131.74} C_VEL
LIN {X 0,Y 538.157,Z 424.073,A -85,B 0,C 180,E1 -4134.755,E2 -4134.755} C_VEL
LIN {X 0,Y 538.162,Z 424.069,A -85,B 0,C 180,E1 -4137.755,E2 -4137.755} C_VEL
LIN {X 0,Y 538.178,Z 424.069,A -85,B 0,C 180,E1 -4140.748,E2 -4140.748} C_VEL
LIN {X 0,Y 538.136,Z 424.074,A -85,B 0,C 180,E1 -4142.995,E2 -4142.995} C_VEL
LIN {X 0,Y 538.126,Z 424.077,A -85,B 0,C 180,E1 -4145.997,E2 -4145.997} C_VEL
LIN {X 0,Y 538.07,Z 424.082,A -85,B 0,C 180,E1 -4149.018,E2 -4149.018} C_VEL
LIN {X 0,Y 538.077,Z 424.083,A -85,B 0,C 180,E1 -4152.063,E2 -4152.063} C_VEL
LIN {X 0,Y 538.039,Z 424.085,A -85,B 0,C 180,E1 -4155.144,E2 -4155.144} C_VEL
LIN {X 0,Y 538.03,Z 424.093,A -85,B 0,C 180,E1 -4158.27,E2 -4158.27} C_VEL
LIN {X 0,Y 538.037,Z 424.091,A -85,B 0,C 180,E1 -4160.652,E2 -4160.652} C_VEL
LIN {X 0,Y 538.018,Z 424.09,A -85,B 0,C 180,E1 -4163.888,E2 -4163.888} C_VEL
LIN {X 0,Y 538.045,Z 424.091,A -85,B 0,C 180,E1 -4166.367,E2 -4166.367} C_VEL
LIN {X 0,Y 538.051,Z 424.085,A -85,B 0,C 180,E1 -4168.939,E2 -4168.939} C_VEL
LIN {X 0,Y 538.023,Z 424.089,A -85,B 0,C 180,E1 -4171.891,E2 -4171.891} C_VEL
LIN {X 0,Y 538.031,Z 424.092,A -85,B 0,C 180,E1 -4174.622,E2 -4174.622} C_VEL
LIN {X 0,Y 538.006,Z 424.092,A -85,B 0,C 180,E1 -4177.172,E2 -4177.172} C_VEL
LIN {X 0,Y 538.044,Z 424.087,A -85,B 0,C 180,E1 -4180.275,E2 -4180.275} C_VEL
LIN {X 0,Y 537.375,Z 424.175,A -85,B 0,C 180,E1 -4180.692,E2 -4180.692} C_VEL
LIN {X 0,Y 534.525,Z 424.528,A -85,B 0,C 180,E1 -4181.343,E2 -4181.343} C_VEL
LIN {X 0,Y 531.657,Z 424.887,A -85,B 0,C 180,E1 -4182.001,E2 -4182.001} C_VEL
LIN {X 0,Y 530.977,Z 424.973,A -85,B 0,C 180,E1 -4182.426,E2 -4182.426} C_VEL
LIN {X 0,Y 531.011,Z 425.099,A -85,B 0,C 180,E1 -4183.49,E2 -4183.49} C_VEL
LIN {X 0,Y 532.784,Z 433.506,A -85,B 0,C 180,E1 -4184.888,E2 -4184.888} C_VEL
LIN {X 0,Y 532.515,Z 446.566,A -85,B 0,C 180,E1 -4186.853,E2 -4186.853} C_VEL
LIN {X 0,Y 535.19,Z 458.74,A -85,B 0,C 180,E1 -4187.138,E2 -4187.138} C_VEL
LIN {X 0,Y 534.318,Z 611.694,A -85,B 0,C 180,E1 -4189.269,E2 -4189.269} C_VEL
LIN {X 0,Y 534.036,Z 626.335,A -85,B 0,C 180,E1 -4189.617,E2 -4189.617} C_VEL
LIN {X 0,Y 533.701,Z 641.144,A -85,B 0,C 180,E1 -4190.124,E2 -4190.124} C_VEL
LIN {X 0,Y 533.295,Z 655.202,A -85,B 0,C 180,E1 -4190.761,E2 -4190.761} C_VEL
LIN {X 0,Y 532.84,Z 669.57,A -85,B 0,C 180,E1 -4191.585,E2 -4191.585} C_VEL
LIN {X 0,Y 532.382,Z 682.873,A -85,B 0,C 180,E1 -4192.529,E2 -4192.529} C_VEL
LIN {X 0,Y 531.984,Z 694.476,A -85,B 0,C 180,E1 -4193.525,E2 -4193.525} C_VEL
LIN {X 0,Y 531.61,Z 705.258,A -85,B 0,C 180,E1 -4194.615,E2 -4194.615} C_VEL
LIN {X 0,Y 531.285,Z 715.135,A -85,B 0,C 180,E1 -4195.793,E2 -4195.793} C_VEL
LIN {X 0,Y 530.996,Z 724.613,A -85,B 0,C 180,E1 -4197.136,E2 -4197.136} C_VEL
LIN {X 0,Y 530.782,Z 732.457,A -85,B 0,C 180,E1 -4198.466,E2 -4198.466} C_VEL
LIN {X 0,Y 530.636,Z 738.953,A -85,B 0,C 180,E1 -4199.783,E2 -4199.783} C_VEL
LIN {X 0,Y 530.527,Z 743.742,A -85,B 0,C 180,E1 -4200.965,E2 -4200.965} C_VEL
LIN {X 0,Y 530.496,Z 748.973,A -85,B 0,C 180,E1 -4202.576,E2 -4202.576} C_VEL
LIN {X 0,Y 530.388,Z 752.979,A -85,B 0,C 180,E1 -4204.297,E2 -4204.297} C_VEL
LIN {X 0,Y 530.358,Z 755.552,A -85,B 0,C 180,E1 -4206.114,E2 -4206.114} C_VEL
LIN {X 0,Y 530.37,Z 756.5,A -85,B 0,C 180,E1 -4208.061,E2 -4208.061} C_VEL
LIN {X 0,Y 530.349,Z 755.689,A -85,B 0,C 180,E1 -4209.847,E2 -4209.847} C_VEL
LIN {X 0,Y 530.369,Z 753.62,A -85,B 0,C 180,E1 -4211.457,E2 -4211.457} C_VEL
LIN {X 0,Y 530.433,Z 750.237,A -85,B 0,C 180,E1 -4213.053,E2 -4213.053} C_VEL
LIN {X 0,Y 530.55,Z 745.506,A -85,B 0,C 180,E1 -4214.638,E2 -4214.638} C_VEL
LIN {X 0,Y 530.628,Z 739.377,A -85,B 0,C 180,E1 -4216.208,E2 -4216.208} C_VEL
LIN {X 0,Y 530.793,Z 731.695,A -85,B 0,C 180,E1 -4217.77,E2 -4217.77} C_VEL
LIN {X 0,Y 531.024,Z 723.489,A -85,B 0,C 180,E1 -4219.13,E2 -4219.13} C_VEL
LIN {X 0,Y 531.318,Z 713.704,A -85,B 0,C 180,E1 -4220.483,E2 -4220.483} C_VEL
LIN {X 0,Y 531.64,Z 703.749,A -85,B 0,C 180,E1 -4221.639,E2 -4221.639} C_VEL
LIN {X 0,Y 532.025,Z 693.315,A -85,B 0,C 180,E1 -4222.67,E2 -4222.67} C_VEL
LIN {X 0,Y 532.467,Z 680.358,A -85,B 0,C 180,E1 -4223.749,E2 -4223.749} C_VEL
LIN {X 0,Y 532.905,Z 667.87,A -85,B 0,C 180,E1 -4224.609,E2 -4224.609} C_VEL
LIN {X 0,Y 533.308,Z 654.344,A -85,B 0,C 180,E1 -4225.371,E2 -4225.371} C_VEL
LIN {X 0,Y 533.702,Z 640.507,A -85,B 0,C 180,E1 -4225.989,E2 -4225.989} C_VEL
LIN {X 0,Y 534.064,Z 625.721,A -85,B 0,C 180,E1 -4226.488,E2 -4226.488} C_VEL
LIN {X 0,Y 534.297,Z 610.485,A -85,B 0,C 180,E1 -4226.843,E2 -4226.843} C_VEL
LIN {X 0,Y 535.162,Z 458.479,A -85,B 0,C 180,E1 -4228.956,E2 -4228.956} C_VEL
LIN {X 0,Y 532.502,Z 446.377,A -85,B 0,C 180,E1 -4229.244,E2 -4229.244} C_VEL
LIN {X 0,Y 532.822,Z 433.884,A -85,B 0,C 180,E1 -4231.134,E2 -4231.134} C_VEL
LIN {X 0,Y 531.115,Z 424.954,A -85,B 0,C 180,E1 -4232.607,E2 -4232.607} C_VEL
LIN {X 0,Y 531.121,Z 424.951,A -85,B 0,C 180,E1 -4235.315,E2 -4235.315} C_VEL
LIN {X 0,Y 531.06,Z 424.957,A -85,B 0,C 180,E1 -4238.371,E2 -4238.371} C_VEL
LIN {X 0,Y 531.072,Z 424.959,A -85,B 0,C 180,E1 -4241.68,E2 -4241.68} C_VEL
LIN {X 0,Y 531.036,Z 424.959,A -85,B 0,C 180,E1 -4244.956,E2 -4244.956} C_VEL
LIN {X 0,Y 531.021,Z 424.966,A -85,B 0,C 180,E1 -4247.722,E2 -4247.722} C_VEL
LIN {X 0,Y 531.004,Z 424.961,A -85,B 0,C 180,E1 -4250.938,E2 -4250.938} C_VEL
LIN {X 0,Y 530.985,Z 424.963,A -85,B 0,C 180,E1 -4254.224,E2 -4254.224} C_VEL
LIN {X 0,Y 531.009,Z 424.96,A -85,B 0,C 180,E1 -4256.744,E2 -4256.744} C_VEL
LIN {X 0,Y 530.986,Z 424.966,A -85,B 0,C 180,E1 -4259.322,E2 -4259.322} C_VEL
LIN {X 0,Y 530.984,Z 424.963,A -85,B 0,C 180,E1 -4262.103,E2 -4262.103} C_VEL
LIN {X 0,Y 530.988,Z 424.963,A -85,B 0,C 180,E1 -4264.853,E2 -4264.853} C_VEL
LIN {X 0,Y 530.97,Z 424.971,A -85,B 0,C 180,E1 -4267.507,E2 -4267.507} C_VEL
LIN {X 0,Y 530.988,Z 424.963,A -85,B 0,C 180,E1 -4270.432,E2 -4270.432} C_VEL
LIN {X 0,Y 530.973,Z 424.967,A -85,B 0,C 180,E1 -4273.282,E2 -4273.282} C_VEL
LIN {X 0,Y 530.99,Z 424.971,A -85,B 0,C 180,E1 -4275.621,E2 -4275.621} C_VEL
LIN {X 0,Y 531.009,Z 424.957,A -85,B 0,C 180,E1 -4278.565,E2 -4278.565} C_VEL
LIN {X 0,Y 530.971,Z 424.969,A -85,B 0,C 180,E1 -4281.346,E2 -4281.346} C_VEL
LIN {X 0,Y 530.984,Z 424.961,A -85,B 0,C 180,E1 -4284.382,E2 -4284.382} C_VEL
LIN {X 0,Y 530.972,Z 424.967,A -85,B 0,C 180,E1 -4287.133,E2 -4287.133} C_VEL
LIN {X 0,Y 530.97,Z 424.968,A -85,B 0,C 180,E1 -4289.803,E2 -4289.803} C_VEL
LIN {X 0,Y 531.019,Z 424.959,A -85,B 0,C 180,E1 -4292.466,E2 -4292.466} C_VEL
LIN {X 0,Y 531.009,Z 424.96,A -85,B 0,C 180,E1 -4294.942,E2 -4294.942} C_VEL
LIN {X 0,Y 530.972,Z 424.965,A -85,B 0,C 180,E1 -4298.246,E2 -4298.246} C_VEL
LIN {X 0,Y 530.996,Z 424.961,A -85,B 0,C 180,E1 -4300.677,E2 -4300.677} C_VEL
LIN {X 0,Y 530.987,Z 424.961,A -85,B 0,C 180,E1 -4303.071,E2 -4303.071} C_VEL
LIN {X 0,Y 531.019,Z 424.962,A -85,B 0,C 180,E1 -4305.436,E2 -4305.436} C_VEL
LIN {X 0,Y 531.037,Z 424.955,A -85,B 0,C 180,E1 -4308.55,E2 -4308.55} C_VEL
LIN {X 0,Y 531.057,Z 424.959,A -85,B 0,C 180,E1 -4311.629,E2 -4311.629} C_VEL
LIN {X 0,Y 531.122,Z 424.945,A -85,B 0,C 180,E1 -4314.685,E2 -4314.685} C_VEL
LIN {X 0,Y 531.139,Z 424.948,A -85,B 0,C 180,E1 -4317.725,E2 -4317.725} C_VEL
LIN {X 0,Y 531.153,Z 424.942,A -85,B 0,C 180,E1 -4320.758,E2 -4320.758} C_VEL
LIN {X 0,Y 531.107,Z 424.947,A -85,B 0,C 180,E1 -4323.034,E2 -4323.034} C_VEL
LIN {X 0,Y 531.083,Z 424.953,A -85,B 0,C 180,E1 -4326.077,E2 -4326.077} C_VEL
LIN {X 0,Y 531.031,Z 424.959,A -85,B 0,C 180,E1 -4329.138,E2 -4329.138} C_VEL
LIN {X 0,Y 531.04,Z 424.954,A -85,B 0,C 180,E1 -4332.225,E2 -4332.225} C_VEL
LIN {X 0,Y 530.995,Z 424.966,A -85,B 0,C 180,E1 -4335.35,E2 -4335.35} C_VEL
LIN {X 0,Y 530.99,Z 424.958,A -85,B 0,C 180,E1 -4338.521,E2 -4338.521} C_VEL
LIN {X 0,Y 530.999,Z 424.961,A -85,B 0,C 180,E1 -4340.938,E2 -4340.938} C_VEL
LIN {X 0,Y 530.979,Z 424.966,A -85,B 0,C 180,E1 -4344.224,E2 -4344.224} C_VEL
LIN {X 0,Y 531.005,Z 424.96,A -85,B 0,C 180,E1 -4346.743,E2 -4346.743} C_VEL
LIN {X 0,Y 530.981,Z 424.967,A -85,B 0,C 180,E1 -4349.323,E2 -4349.323} C_VEL
LIN {X 0,Y 530.969,Z 424.969,A -85,B 0,C 180,E1 -4352.101,E2 -4352.101} C_VEL
LIN {X 0,Y 530.989,Z 424.963,A -85,B 0,C 180,E1 -4354.854,E2 -4354.854} C_VEL
LIN {X 0,Y 530.966,Z 424.972,A -85,B 0,C 180,E1 -4357.507,E2 -4357.507} C_VEL
LIN {X 0,Y 530.983,Z 424.964,A -85,B 0,C 180,E1 -4360.433,E2 -4360.433} C_VEL
LIN {X 0,Y 530.963,Z 424.969,A -85,B 0,C 180,E1 -4363.281,E2 -4363.281} C_VEL
LIN {X 0,Y 530.988,Z 424.971,A -85,B 0,C 180,E1 -4365.621,E2 -4365.621} C_VEL
LIN {X 0,Y 530.997,Z 424.963,A -85,B 0,C 180,E1 -4368.565,E2 -4368.565} C_VEL
LIN {X 0,Y 530.959,Z 424.974,A -85,B 0,C 180,E1 -4371.529,E2 -4371.529} C_VEL
LIN {X 0,Y 530.954,Z 424.971,A -85,B 0,C 180,E1 -4374.38,E2 -4374.38} C_VEL
LIN {X 0,Y 530.968,Z 424.97,A -85,B 0,C 180,E1 -4377.133,E2 -4377.133} C_VEL
LIN {X 0,Y 530.971,Z 424.974,A -85,B 0,C 180,E1 -4379.803,E2 -4379.803} C_VEL
LIN {X 0,Y 531.023,Z 424.972,A -85,B 0,C 180,E1 -4382.183,E2 -4382.183} C_VEL
LIN {X 0,Y 533.741,Z 437.008,A -85,B 0,C 180,E1 -4383.94,E2 -4383.94} C_VEL
LIN {X 0,Y 533.132,Z 458.228,A -85,B 0,C 180,E1 -4386.704,E2 -4386.704} C_VEL
LIN {X 0,Y 532.682,Z 474.512,A -85,B 0,C 180,E1 -4388.797,E2 -4388.797} C_VEL
LIN {X 0,Y 535.151,Z 487.011,A -85,B 0,C 180,E1 -4389.078,E2 -4389.078} C_VEL
LIN {X 0,Y 534.281,Z 640.45,A -85,B 0,C 180,E1 -4391.207,E2 -4391.207} C_VEL
LIN {X 0,Y 534.045,Z 656.49,A -85,B 0,C 180,E1 -4391.588,E2 -4391.588} C_VEL
LIN {X 0,Y 533.712,Z 670.638,A -85,B 0,C 180,E1 -4392.073,E2 -4392.073} C_VEL
LIN {X 0,Y 533.343,Z 683.687,A -85,B 0,C 180,E1 -4392.654,E2 -4392.654} C_VEL
LIN {X 0,Y 532.885,Z 697.622,A -85,B 0,C 180,E1 -4393.429,E2 -4393.429} C_VEL
LIN {X 0,Y 532.493,Z 710.378,A -85,B 0,C 180,E1 -4394.302,E2 -4394.302} C_VEL
LIN {X 0,Y 532.04,Z 723.215,A -85,B 0,C 180,E1 -4395.366,E2 -4395.366} C_VEL
LIN {X 0,Y 531.648,Z 733.962,A -85,B 0,C 180,E1 -4396.429,E2 -4396.429} C_VEL
LIN {X 0,Y 531.314,Z 743.901,A -85,B 0,C 180,E1 -4397.587,E2 -4397.587} C_VEL
LIN {X 0,Y 531.081,Z 753.62,A -85,B 0,C 180,E1 -4398.937,E2 -4398.937} C_VEL
LIN {X 0,Y 530.78,Z 761.724,A -85,B 0,C 180,E1 -4400.28,E2 -4400.28} C_VEL
LIN {X 0,Y 530.665,Z 768.421,A -85,B 0,C 180,E1 -4401.623,E2 -4401.623} C_VEL
LIN {X 0,Y 530.549,Z 774.604,A -85,B 0,C 180,E1 -4403.153,E2 -4403.153} C_VEL
LIN {X 0,Y 530.508,Z 779.385,A -85,B 0,C 180,E1 -4404.679,E2 -4404.679} C_VEL
LIN {X 0,Y 530.481,Z 782.886,A -85,B 0,C 180,E1 -4406.201,E2 -4406.201} C_VEL
LIN {X 0,Y 530.407,Z 785.189,A -85,B 0,C 180,E1 -4407.721,E2 -4407.721} C_VEL
LIN {X 0,Y 530.341,Z 786.348,A -85,B 0,C 180,E1 -4409.24,E2 -4409.24} C_VEL
LIN {X 0,Y 530.341,Z 786.347,A -85,B 0,C 180,E1 -4410.759,E2 -4410.759} C_VEL
LIN {X 0,Y 530.407,Z 785.187,A -85,B 0,C 180,E1 -4412.278,E2 -4412.278} C_VEL
LIN {X 0,Y 530.48,Z 782.884,A -85,B 0,C 180,E1 -4413.798,E2 -4413.798} C_VEL
LIN {X 0,Y 530.508,Z 779.388,A -85,B 0,C 180,E1 -4415.32,E2 -4415.32} C_VEL
LIN {X 0,Y 530.549,Z 774.611,A -85,B 0,C 180,E1 -4416.847,E2 -4416.847} C_VEL
LIN {X 0,Y 530.665,Z 768.422,A -85,B 0,C 180,E1 -4418.376,E2 -4418.376} C_VEL
LIN {X 0,Y 530.809,Z 760.646,A -85,B 0,C 180,E1 -4419.911,E2 -4419.911} C_VEL
LIN {X 0,Y 531.056,Z 752.37,A -85,B 0,C 180,E1 -4421.256,E2 -4421.256} C_VEL
LIN {X 0,Y 531.382,Z 742.396,A -85,B 0,C 180,E1 -4422.604,E2 -4422.604} C_VEL
LIN {X 0,Y 531.709,Z 732.189,A -85,B 0,C 180,E1 -4423.763,E2 -4423.763} C_VEL
LIN {X 0,Y 532.12,Z 720.024,A -85,B 0,C 180,E1 -4424.924,E2 -4424.924} C_VEL
LIN {X 0,Y 532.593,Z 706.596,A -85,B 0,C 180,E1 -4425.98,E2 -4425.98} C_VEL
LIN {X 0,Y 533.08,Z 692.821,A -85,B 0,C 180,E1 -4426.86,E2 -4426.86} C_VEL
LIN {X 0,Y 533.457,Z 678.679,A -85,B 0,C 180,E1 -4427.588,E2 -4427.588} C_VEL
LIN {X 0,Y 533.819,Z 664.13,A -85,B 0,C 180,E1 -4428.171,E2 -4428.171} C_VEL
LIN {X 0,Y 534.153,Z 648.371,A -85,B 0,C 180,E1 -4428.627,E2 -4428.627} C_VEL
LIN {X 0,Y 534.369,Z 632.156,A -85,B 0,C 180,E1 -4428.923,E2 -4428.923} C_VEL
LIN {X 0,Y 535.168,Z 486.988,A -85,B 0,C 180,E1 -4430.921,E2 -4430.921} C_VEL
LIN {X 0,Y 532.682,Z 474.4,A -85,B 0,C 180,E1 -4431.21,E2 -4431.21} C_VEL
LIN {X 0,Y 533.286,Z 451.823,A -85,B 0,C 180,E1 -4434.112,E2 -4434.112} C_VEL
LIN {X 0,Y 533.69,Z 436.89,A -85,B 0,C 180,E1 -4436.059,E2 -4436.059} C_VEL
LIN {X 0,Y 531.022,Z 424.972,A -85,B 0,C 180,E1 -4437.816,E2 -4437.816} C_VEL
LIN {X 0,Y 530.979,Z 424.971,A -85,B 0,C 180,E1 -4440.646,E2 -4440.646} C_VEL
LIN {X 0,Y 530.986,Z 424.967,A -85,B 0,C 180,E1 -4443.772,E2 -4443.772} C_VEL
LIN {X 0,Y 530.965,Z 424.971,A -85,B 0,C 180,E1 -4446.557,E2 -4446.557} C_VEL
LIN {X 0,Y 531.002,Z 424.965,A -85,B 0,C 180,E1 -4449.857,E2 -4449.857} C_VEL
LIN {X 0,Y 530.979,Z 424.969,A -85,B 0,C 180,E1 -4452.455,E2 -4452.455} C_VEL
LIN {X 0,Y 530.98,Z 424.966,A -85,B 0,C 180,E1 -4455.62,E2 -4455.62} C_VEL
LIN {X 0,Y 530.995,Z 424.968,A -85,B 0,C 180,E1 -4458.565,E2 -4458.565} C_VEL
LIN {X 0,Y 530.953,Z 424.968,A -85,B 0,C 180,E1 -4461.529,E2 -4461.529} C_VEL
LIN {X 0,Y 530.977,Z 424.972,A -85,B 0,C 180,E1 -4464.382,E2 -4464.382} C_VEL
LIN {X 0,Y 530.969,Z 424.965,A -85,B 0,C 180,E1 -4467.134,E2 -4467.134} C_VEL
LIN {X 0,Y 530.963,Z 424.968,A -85,B 0,C 180,E1 -4469.803,E2 -4469.803} C_VEL
LIN {X 0,Y 531.011,Z 424.966,A -85,B 0,C 180,E1 -4472.466,E2 -4472.466} C_VEL
LIN {X 0,Y 531.001,Z 424.962,A -85,B 0,C 180,E1 -4474.942,E2 -4474.942} C_VEL
LIN {X 0,Y 530.964,Z 424.974,A -85,B 0,C 180,E1 -4478.247,E2 -4478.247} C_VEL
LIN {X 0,Y 530.99,Z 424.967,A -85,B 0,C 180,E1 -4480.677,E2 -4480.677} C_VEL
LIN {X 0,Y 530.985,Z 424.962,A -85,B 0,C 180,E1 -4483.071,E2 -4483.071} C_VEL
LIN {X 0,Y 531.011,Z 424.96,A -85,B 0,C 180,E1 -4485.436,E2 -4485.436} C_VEL
LIN {X 0,Y 531.041,Z 424.962,A -85,B 0,C 180,E1 -4488.55,E2 -4488.55} C_VEL
LIN {X 0,Y 531.053,Z 424.955,A -85,B 0,C 180,E1 -4491.63,E2 -4491.63} C_VEL
LIN {X 0,Y 531.116,Z 424.951,A -85,B 0,C 180,E1 -4494.685,E2 -4494.685} C_VEL
LIN {X 0,Y 531.134,Z 424.944,A -85,B 0,C 180,E1 -4497.725,E2 -4497.725} C_VEL
LIN {X 0,Y 531.148,Z 424.944,A -85,B 0,C 180,E1 -4500.758,E2 -4500.758} C_VEL
LIN {X 0,Y 531.102,Z 424.95,A -85,B 0,C 180,E1 -4503.034,E2 -4503.034} C_VEL
LIN {X 0,Y 531.084,Z 424.955,A -85,B 0,C 180,E1 -4506.077,E2 -4506.077} C_VEL
LIN {X 0,Y 531.029,Z 424.959,A -85,B 0,C 180,E1 -4509.138,E2 -4509.138} C_VEL
LIN {X 0,Y 531.034,Z 424.963,A -85,B 0,C 180,E1 -4512.225,E2 -4512.225} C_VEL
LIN {X 0,Y 530.99,Z 424.963,A -85,B 0,C 180,E1 -4515.35,E2 -4515.35} C_VEL
LIN {X 0,Y 531.01,Z 424.961,A -85,B 0,C 180,E1 -4517.723,E2 -4517.723} C_VEL
LIN {X 0,Y 530.996,Z 424.964,A -85,B 0,C 180,E1 -4520.938,E2 -4520.938} C_VEL
LIN {X 0,Y 530.974,Z 424.972,A -85,B 0,C 180,E1 -4524.225,E2 -4524.225} C_VEL
LIN {X 0,Y 531.007,Z 424.966,A -85,B 0,C 180,E1 -4526.744,E2 -4526.744} C_VEL
LIN {X 0,Y 530.995,Z 424.962,A -85,B 0,C 180,E1 -4529.322,E2 -4529.322} C_VEL
LIN {X 0,Y 530.976,Z 424.97,A -85,B 0,C 180,E1 -4532.104,E2 -4532.104} C_VEL
LIN {X 0,Y 530.987,Z 424.968,A -85,B 0,C 180,E1 -4534.855,E2 -4534.855} C_VEL
LIN {X 0,Y 530.964,Z 424.969,A -85,B 0,C 180,E1 -4537.508,E2 -4537.508} C_VEL
LIN {X 0,Y 531.023,Z 424.967,A -85,B 0,C 180,E1 -4540.429,E2 -4540.429} C_VEL
LIN {X 0,Y 530.977,Z 424.973,A -85,B 0,C 180,E1 -4542.426,E2 -4542.426} C_VEL
LIN {X 0,Y 530.756,Z 425.367,A -85,B 0,C 180,E1 -4542.844,E2 -4542.844} C_VEL
LIN {X 0,Y 529.829,Z 427.12,A -85,B 0,C 180,E1 -4543.444,E2 -4543.444} C_VEL
LIN {X 0,Y 528.545,Z 429.823,A -85,B 0,C 180,E1 -4544,E2 -4544} C_VEL
LIN {X 0,Y 526.808,Z 434.397,A -85,B 0,C 180,E1 -4544.716,E2 -4544.716} C_VEL
LIN {X 0,Y 525.874,Z 439.256,A -85,B 0,C 180,E1 -4545.427,E2 -4545.427} C_VEL
LIN {X 0,Y 525.704,Z 446.886,A -85,B 0,C 180,E1 -4546.566,E2 -4546.566} C_VEL
LIN {X 0,Y 528.62,Z 460.5,A -85,B 0,C 180,E1 -4546.888,E2 -4546.888} C_VEL
LIN {X 0,Y 527.619,Z 611.71,A -85,B 0,C 180,E1 -4549.02,E2 -4549.02} C_VEL
LIN {X 0,Y 527.319,Z 626.574,A -85,B 0,C 180,E1 -4549.377,E2 -4549.377} C_VEL
LIN {X 0,Y 526.942,Z 641.563,A -85,B 0,C 180,E1 -4549.897,E2 -4549.897} C_VEL
LIN {X 0,Y 526.497,Z 656.619,A -85,B 0,C 180,E1 -4550.595,E2 -4550.595} C_VEL
LIN {X 0,Y 526.021,Z 669.466,A -85,B 0,C 180,E1 -4551.347,E2 -4551.347} C_VEL
LIN {X 0,Y 525.529,Z 682.516,A -85,B 0,C 180,E1 -4552.28,E2 -4552.28} C_VEL
LIN {X 0,Y 525.109,Z 693.757,A -85,B 0,C 180,E1 -4553.246,E2 -4553.246} C_VEL
LIN {X 0,Y 524.671,Z 704.743,A -85,B 0,C 180,E1 -4554.361,E2 -4554.361} C_VEL
LIN {X 0,Y 524.325,Z 714.312,A -85,B 0,C 180,E1 -4555.507,E2 -4555.507} C_VEL
LIN {X 0,Y 523.989,Z 723.887,A -85,B 0,C 180,E1 -4556.87,E2 -4556.87} C_VEL
LIN {X 0,Y 523.772,Z 731.046,A -85,B 0,C 180,E1 -4558.07,E2 -4558.07} C_VEL
LIN {X 0,Y 523.578,Z 738.425,A -85,B 0,C 180,E1 -4559.555,E2 -4559.555} C_VEL
LIN {X 0,Y 523.447,Z 744.579,A -85,B 0,C 180,E1 -4561.096,E2 -4561.096} C_VEL
LIN {X 0,Y 523.4,Z 748.701,A -85,B 0,C 180,E1 -4562.403,E2 -4562.403} C_VEL
LIN {X 0,Y 523.284,Z 752.777,A -85,B 0,C 180,E1 -4564.139,E2 -4564.139} C_VEL
LIN {X 0,Y 523.251,Z 754.804,A -85,B 0,C 180,E1 -4565.395,E2 -4565.395} C_VEL
LIN {X 0,Y 523.242,Z 756.262,A -85,B 0,C 180,E1 -4567.076,E2 -4567.076} C_VEL
LIN {X 0,Y 523.265,Z 756.363,A -85,B 0,C 180,E1 -4568.738,E2 -4568.738} C_VEL
LIN {X 0,Y 523.287,Z 755.16,A -85,B 0,C 180,E1 -4570.382,E2 -4570.382} C_VEL
LIN {X 0,Y 523.287,Z 752.675,A -85,B 0,C 180,E1 -4572.008,E2 -4572.008} C_VEL
LIN {X 0,Y 523.375,Z 748.881,A -85,B 0,C 180,E1 -4573.621,E2 -4573.621} C_VEL
LIN {X 0,Y 523.511,Z 743.731,A -85,B 0,C 180,E1 -4575.223,E2 -4575.223} C_VEL
LIN {X 0,Y 523.606,Z 737.143,A -85,B 0,C 180,E1 -4576.811,E2 -4576.811} C_VEL
LIN {X 0,Y 523.89,Z 728.912,A -85,B 0,C 180,E1 -4578.392,E2 -4578.392} C_VEL
LIN {X 0,Y 524.113,Z 720.246,A -85,B 0,C 180,E1 -4579.766,E2 -4579.766} C_VEL
LIN {X 0,Y 524.461,Z 709.88,A -85,B 0,C 180,E1 -4581.136,E2 -4581.136} C_VEL
LIN {X 0,Y 524.889,Z 699.279,A -85,B 0,C 180,E1 -4582.306,E2 -4582.306} C_VEL
LIN {X 0,Y 525.371,Z 686.635,A -85,B 0,C 180,E1 -4583.471,E2 -4583.471} C_VEL
LIN {X 0,Y 525.84,Z 673.937,A -85,B 0,C 180,E1 -4584.44,E2 -4584.44} C_VEL
LIN {X 0,Y 526.376,Z 659.943,A -85,B 0,C 180,E1 -4585.31,E2 -4585.31} C_VEL
LIN {X 0,Y 526.813,Z 645.306,A -85,B 0,C 180,E1 -4586.032,E2 -4586.032} C_VEL
LIN {X 0,Y 527.214,Z 630.583,A -85,B 0,C 180,E1 -4586.585,E2 -4586.585} C_VEL
LIN {X 0,Y 527.493,Z 615.374,A -85,B 0,C 180,E1 -4586.993,E2 -4586.993} C_VEL
LIN {X 0,Y 527.68,Z 595.451,A -85,B 0,C 180,E1 -4587.319,E2 -4587.319} C_VEL
LIN {X 0,Y 528.515,Z 459.376,A -85,B 0,C 180,E1 -4589.221,E2 -4589.221} C_VEL
LIN {X 0,Y 525.644,Z 446.598,A -85,B 0,C 180,E1 -4589.532,E2 -4589.532} C_VEL
LIN {X 0,Y 525.898,Z 434.831,A -85,B 0,C 180,E1 -4591.34,E2 -4591.34} C_VEL
LIN {X 0,Y 524.064,Z 425.833,A -85,B 0,C 180,E1 -4592.859,E2 -4592.859} C_VEL
LIN {X 0,Y 524.031,Z 425.835,A -85,B 0,C 180,E1 -4596.16,E2 -4596.16} C_VEL
LIN {X 0,Y 524.008,Z 425.835,A -85,B 0,C 180,E1 -4598.484,E2 -4598.484} C_VEL
LIN {X 0,Y 524.03,Z 425.837,A -85,B 0,C 180,E1 -4601.751,E2 -4601.751} C_VEL
LIN {X 0,Y 523.998,Z 425.836,A -85,B 0,C 180,E1 -4605.053,E2 -4605.053} C_VEL
LIN {X 0,Y 523.968,Z 425.842,A -85,B 0,C 180,E1 -4607.969,E2 -4607.969} C_VEL
LIN {X 0,Y 523.977,Z 425.837,A -85,B 0,C 180,E1 -4610.41,E2 -4610.41} C_VEL
LIN {X 0,Y 523.922,Z 425.845,A -85,B 0,C 180,E1 -4612.893,E2 -4612.893} C_VEL
LIN {X 0,Y 523.958,Z 425.843,A -85,B 0,C 180,E1 -4615.419,E2 -4615.419} C_VEL
LIN {X 0,Y 523.974,Z 425.839,A -85,B 0,C 180,E1 -4617.999,E2 -4617.999} C_VEL
LIN {X 0,Y 523.951,Z 425.84,A -85,B 0,C 180,E1 -4620.855,E2 -4620.855} C_VEL
LIN {X 0,Y 523.964,Z 425.845,A -85,B 0,C 180,E1 -4623.735,E2 -4623.735} C_VEL
LIN {X 0,Y 523.925,Z 425.842,A -85,B 0,C 180,E1 -4626.404,E2 -4626.404} C_VEL
LIN {X 0,Y 523.926,Z 425.841,A -85,B 0,C 180,E1 -4629.084,E2 -4629.084} C_VEL
LIN {X 0,Y 523.96,Z 425.839,A -85,B 0,C 180,E1 -4632.118,E2 -4632.118} C_VEL
LIN {X 0,Y 523.958,Z 425.842,A -85,B 0,C 180,E1 -4635.308,E2 -4635.308} C_VEL
LIN {X 0,Y 523.974,Z 425.833,A -85,B 0,C 180,E1 -4638.687,E2 -4638.687} C_VEL
LIN {X 0,Y 523.927,Z 425.844,A -85,B 0,C 180,E1 -4641.079,E2 -4641.079} C_VEL
LIN {X 0,Y 523.932,Z 425.845,A -85,B 0,C 180,E1 -4643.827,E2 -4643.827} C_VEL
LIN {X 0,Y 523.944,Z 425.84,A -85,B 0,C 180,E1 -4646.635,E2 -4646.635} C_VEL
LIN {X 0,Y 523.956,Z 425.842,A -85,B 0,C 180,E1 -4649.355,E2 -4649.355} C_VEL
LIN {X 0,Y 523.982,Z 425.837,A -85,B 0,C 180,E1 -4652.28,E2 -4652.28} C_VEL
LIN {X 0,Y 523.956,Z 425.838,A -85,B 0,C 180,E1 -4654.581,E2 -4654.581} C_VEL
LIN {X 0,Y 523.912,Z 425.84,A -85,B 0,C 180,E1 -4657.106,E2 -4657.106} C_VEL
LIN {X 0,Y 523.979,Z 425.842,A -85,B 0,C 180,E1 -4659.866,E2 -4659.866} C_VEL
LIN {X 0,Y 523.968,Z 425.834,A -85,B 0,C 180,E1 -4662.837,E2 -4662.837} C_VEL
LIN {X 0,Y 523.977,Z 425.836,A -85,B 0,C 180,E1 -4665.235,E2 -4665.235} C_VEL
LIN {X 0,Y 524.012,Z 425.83,A -85,B 0,C 180,E1 -4668.394,E2 -4668.394} C_VEL
LIN {X 0,Y 524.005,Z 425.835,A -85,B 0,C 180,E1 -4671.516,E2 -4671.516} C_VEL
LIN {X 0,Y 524.083,Z 425.822,A -85,B 0,C 180,E1 -4674.613,E2 -4674.613} C_VEL
LIN {X 0,Y 524.111,Z 425.823,A -85,B 0,C 180,E1 -4677.694,E2 -4677.694} C_VEL
LIN {X 0,Y 524.124,Z 425.818,A -85,B 0,C 180,E1 -4680.768,E2 -4680.768} C_VEL
LIN {X 0,Y 524.073,Z 425.823,A -85,B 0,C 180,E1 -4683.075,E2 -4683.075} C_VEL
LIN {X 0,Y 524.045,Z 425.829,A -85,B 0,C 180,E1 -4686.159,E2 -4686.159} C_VEL
LIN {X 0,Y 523.999,Z 425.836,A -85,B 0,C 180,E1 -4689.262,E2 -4689.262} C_VEL
LIN {X 0,Y 524.002,Z 425.835,A -85,B 0,C 180,E1 -4691.739,E2 -4691.739} C_VEL
LIN {X 0,Y 523.992,Z 425.835,A -85,B 0,C 180,E1 -4695.052,E2 -4695.052} C_VEL
LIN {X 0,Y 523.963,Z 425.838,A -85,B 0,C 180,E1 -4697.969,E2 -4697.969} C_VEL
LIN {X 0,Y 523.971,Z 425.837,A -85,B 0,C 180,E1 -4700.41,E2 -4700.41} C_VEL
LIN {X 0,Y 523.916,Z 425.843,A -85,B 0,C 180,E1 -4702.893,E2 -4702.893} C_VEL
LIN {X 0,Y 523.952,Z 425.844,A -85,B 0,C 180,E1 -4705.419,E2 -4705.419} C_VEL
LIN {X 0,Y 523.97,Z 425.841,A -85,B 0,C 180,E1 -4707.999,E2 -4707.999} C_VEL
LIN {X 0,Y 523.944,Z 425.84,A -85,B 0,C 180,E1 -4710.855,E2 -4710.855} C_VEL
LIN {X 0,Y 523.961,Z 425.846,A -85,B 0,C 180,E1 -4713.735,E2 -4713.735} C_VEL
LIN {X 0,Y 523.922,Z 425.844,A -85,B 0,C 180,E1 -4716.404,E2 -4716.404} C_VEL
LIN {X 0,Y 523.922,Z 425.844,A -85,B 0,C 180,E1 -4719.084,E2 -4719.084} C_VEL
LIN {X 0,Y 523.953,Z 425.843,A -85,B 0,C 180,E1 -4722.119,E2 -4722.119} C_VEL
LIN {X 0,Y 523.956,Z 425.842,A -85,B 0,C 180,E1 -4725.309,E2 -4725.309} C_VEL
LIN {X 0,Y 523.959,Z 425.839,A -85,B 0,C 180,E1 -4728.689,E2 -4728.689} C_VEL
LIN {X 0,Y 523.918,Z 425.846,A -85,B 0,C 180,E1 -4731.08,E2 -4731.08} C_VEL
LIN {X 0,Y 523.9,Z 425.853,A -85,B 0,C 180,E1 -4733.825,E2 -4733.825} C_VEL
LIN {X 0,Y 523.941,Z 425.844,A -85,B 0,C 180,E1 -4736.636,E2 -4736.636} C_VEL
LIN {X 0,Y 523.957,Z 425.846,A -85,B 0,C 180,E1 -4739.356,E2 -4739.356} C_VEL
LIN {X 0,Y 524.025,Z 426.04,A -85,B 0,C 180,E1 -4741.95,E2 -4741.95} C_VEL
LIN {X 0,Y 526.928,Z 439.117,A -85,B 0,C 180,E1 -4743.887,E2 -4743.887} C_VEL
LIN {X 0,Y 526.194,Z 461.508,A -85,B 0,C 180,E1 -4746.837,E2 -4746.837} C_VEL
LIN {X 0,Y 525.834,Z 474.419,A -85,B 0,C 180,E1 -4748.512,E2 -4748.512} C_VEL
LIN {X 0,Y 528.557,Z 488.641,A -85,B 0,C 180,E1 -4748.831,E2 -4748.831} C_VEL
LIN {X 0,Y 527.544,Z 641.217,A -85,B 0,C 180,E1 -4750.979,E2 -4750.979} C_VEL
LIN {X 0,Y 527.287,Z 656.229,A -85,B 0,C 180,E1 -4751.344,E2 -4751.344} C_VEL
LIN {X 0,Y 526.919,Z 670.387,A -85,B 0,C 180,E1 -4751.834,E2 -4751.834} C_VEL
LIN {X 0,Y 526.505,Z 683.447,A -85,B 0,C 180,E1 -4752.422,E2 -4752.422} C_VEL
LIN {X 0,Y 526.027,Z 697.389,A -85,B 0,C 180,E1 -4753.206,E2 -4753.206} C_VEL
LIN {X 0,Y 525.591,Z 710.681,A -85,B 0,C 180,E1 -4754.13,E2 -4754.13} C_VEL
LIN {X 0,Y 525.049,Z 723.085,A -85,B 0,C 180,E1 -4755.168,E2 -4755.168} C_VEL
LIN {X 0,Y 524.677,Z 733.886,A -85,B 0,C 180,E1 -4756.245,E2 -4756.245} C_VEL
LIN {X 0,Y 524.336,Z 743.891,A -85,B 0,C 180,E1 -4757.419,E2 -4757.419} C_VEL
LIN {X 0,Y 524.051,Z 753.619,A -85,B 0,C 180,E1 -4758.787,E2 -4758.787} C_VEL
LIN {X 0,Y 523.739,Z 761.725,A -85,B 0,C 180,E1 -4760.148,E2 -4760.148} C_VEL
LIN {X 0,Y 523.612,Z 768.421,A -85,B 0,C 180,E1 -4761.509,E2 -4761.509} C_VEL
LIN {X 0,Y 523.481,Z 774.604,A -85,B 0,C 180,E1 -4763.06,E2 -4763.06} C_VEL
LIN {X 0,Y 523.441,Z 779.385,A -85,B 0,C 180,E1 -4764.607,E2 -4764.607} C_VEL
LIN {X 0,Y 523.402,Z 782.886,A -85,B 0,C 180,E1 -4766.15,E2 -4766.15} C_VEL
LIN {X 0,Y 523.331,Z 785.189,A -85,B 0,C 180,E1 -4767.691,E2 -4767.691} C_VEL
LIN {X 0,Y 523.247,Z 786.347,A -85,B 0,C 180,E1 -4769.23,E2 -4769.23} C_VEL
LIN {X 0,Y 523.247,Z 786.347,A -85,B 0,C 180,E1 -4770.769,E2 -4770.769} C_VEL
LIN {X 0,Y 523.331,Z 785.186,A -85,B 0,C 180,E1 -4772.309,E2 -4772.309} C_VEL
LIN {X 0,Y 523.402,Z 782.883,A -85,B 0,C 180,E1 -4773.849,E2 -4773.849} C_VEL
LIN {X 0,Y 523.441,Z 779.388,A -85,B 0,C 180,E1 -4775.392,E2 -4775.392} C_VEL
LIN {X 0,Y 523.48,Z 774.611,A -85,B 0,C 180,E1 -4776.939,E2 -4776.939} C_VEL
LIN {X 0,Y 523.611,Z 768.422,A -85,B 0,C 180,E1 -4778.49,E2 -4778.49} C_VEL
LIN {X 0,Y 523.775,Z 760.645,A -85,B 0,C 180,E1 -4780.045,E2 -4780.045} C_VEL
LIN {X 0,Y 524.017,Z 752.37,A -85,B 0,C 180,E1 -4781.409,E2 -4781.409} C_VEL
LIN {X 0,Y 524.379,Z 742.374,A -85,B 0,C 180,E1 -4782.775,E2 -4782.775} C_VEL
LIN {X 0,Y 524.746,Z 732.097,A -85,B 0,C 180,E1 -4783.949,E2 -4783.949} C_VEL
LIN {X 0,Y 525.204,Z 719.854,A -85,B 0,C 180,E1 -4785.125,E2 -4785.125} C_VEL
LIN {X 0,Y 525.701,Z 706.228,A -85,B 0,C 180,E1 -4786.204,E2 -4786.204} C_VEL
LIN {X 0,Y 526.225,Z 692.565,A -85,B 0,C 180,E1 -4787.086,E2 -4787.086} C_VEL
LIN {X 0,Y 526.666,Z 678.415,A -85,B 0,C 180,E1 -4787.823,E2 -4787.823} C_VEL
LIN {X 0,Y 527.061,Z 663.854,A -85,B 0,C 180,E1 -4788.412,E2 -4788.412} C_VEL
LIN {X 0,Y 527.39,Z 648.063,A -85,B 0,C 180,E1 -4788.875,E2 -4788.875} C_VEL
LIN {X 0,Y 527.651,Z 632.832,A -85,B 0,C 180,E1 -4789.159,E2 -4789.159} C_VEL
LIN {X 0,Y 528.552,Z 488.15,A -85,B 0,C 180,E1 -4791.175,E2 -4791.175} C_VEL
LIN {X 0,Y 525.804,Z 474.097,A -85,B 0,C 180,E1 -4791.51,E2 -4791.51} C_VEL
LIN {X 0,Y 526.492,Z 451.614,A -85,B 0,C 180,E1 -4794.444,E2 -4794.444} C_VEL
LIN {X 0,Y 526.871,Z 438.961,A -85,B 0,C 180,E1 -4796.115,E2 -4796.115} C_VEL
LIN {X 0,Y 523.998,Z 425.846,A -85,B 0,C 180,E1 -4798.078,E2 -4798.078} C_VEL
LIN {X 0,Y 523.949,Z 425.845,A -85,B 0,C 180,E1 -4800.856,E2 -4800.856} C_VEL
LIN {X 0,Y 523.957,Z 425.842,A -85,B 0,C 180,E1 -4803.734,E2 -4803.734} C_VEL
LIN {X 0,Y 523.919,Z 425.851,A -85,B 0,C 180,E1 -4806.404,E2 -4806.404} C_VEL
LIN {X 0,Y 523.956,Z 425.84,A -85,B 0,C 180,E1 -4809.081,E2 -4809.081} C_VEL
LIN {X 0,Y 523.953,Z 425.847,A -85,B 0,C 180,E1 -4812.118,E2 -4812.118} C_VEL
LIN {X 0,Y 523.949,Z 425.841,A -85,B 0,C 180,E1 -4815.308,E2 -4815.308} C_VEL
LIN {X 0,Y 523.956,Z 425.843,A -85,B 0,C 180,E1 -4818.688,E2 -4818.688} C_VEL
LIN {X 0,Y 523.911,Z 425.848,A -85,B 0,C 180,E1 -4821.898,E2 -4821.898} C_VEL
LIN {X 0,Y 523.933,Z 425.844,A -85,B 0,C 180,E1 -4824.908,E2 -4824.908} C_VEL
LIN {X 0,Y 523.937,Z 425.841,A -85,B 0,C 180,E1 -4827.678,E2 -4827.678} C_VEL
LIN {X 0,Y 523.948,Z 425.844,A -85,B 0,C 180,E1 -4830.676,E2 -4830.676} C_VEL
LIN {X 0,Y 523.971,Z 425.837,A -85,B 0,C 180,E1 -4833.729,E2 -4833.729} C_VEL
LIN {X 0,Y 523.929,Z 425.849,A -85,B 0,C 180,E1 -4836.271,E2 -4836.271} C_VEL
LIN {X 0,Y 523.94,Z 425.842,A -85,B 0,C 180,E1 -4838.767,E2 -4838.767} C_VEL
LIN {X 0,Y 523.947,Z 425.84,A -85,B 0,C 180,E1 -4841.221,E2 -4841.221} C_VEL
